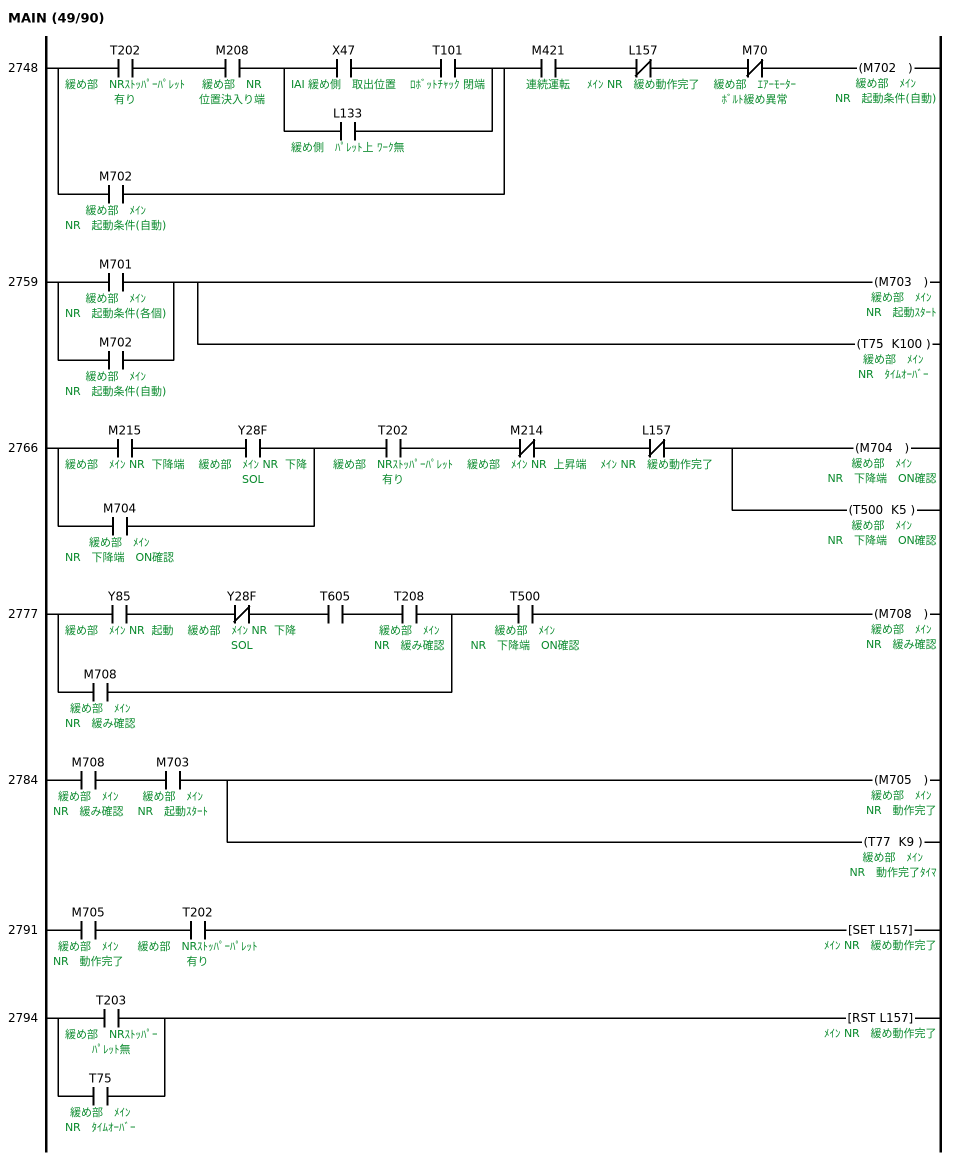
[picture p48: ladder of MAIN, rungs at steps 2748 to 2794]
2748  LD      T202  ; 緩め部　NRｽﾄｯﾊﾟｰﾊﾟﾚｯﾄ有り
      AND     M208  ; 緩め部　NR 位置決入り端
      LD      X47  ; IAI 緩め側　取出位置
      AND     T101  ; ﾛﾎﾞｯﾄﾁｬｯｸ 閉端
      OR      L133  ; 緩め側　ﾊﾟﾚｯﾄ上 ﾜｰｸ無
      ANB
      OR      M702  ; 緩め部　ﾒｲﾝ NR　起動条件(自動)
      AND     M421  ; 連続運転
      ANI     L157  ; ﾒｲﾝ NR　緩め動作完了
      ANI     M70  ; 緩め部　ｴｱｰﾓｰﾀｰ ﾎﾞﾙﾄ緩め異常
      OUT     M702  ; 緩め部　ﾒｲﾝ NR　起動条件(自動)
2759  LD      M701  ; 緩め部　ﾒｲﾝ NR　起動条件(各個)
      OR      M702  ; 緩め部　ﾒｲﾝ NR　起動条件(自動)
      OUT     M703  ; 緩め部　ﾒｲﾝ NR　起動ｽﾀｰﾄ
      OUT     T75 K100  ; 緩め部　ﾒｲﾝ NR　ﾀｲﾑｵｰﾊﾞｰ
2766  LD      M215  ; 緩め部　ﾒｲﾝ NR  下降端
      AND     Y28F  ; 緩め部　ﾒｲﾝ NR  下降 SOL
      OR      M704  ; 緩め部　ﾒｲﾝ NR　下降端　ON確認
      AND     T202  ; 緩め部　NRｽﾄｯﾊﾟｰﾊﾟﾚｯﾄ有り
      ANI     M214  ; 緩め部　ﾒｲﾝ NR  上昇端
      ANI     L157  ; ﾒｲﾝ NR　緩め動作完了
      OUT     M704  ; 緩め部　ﾒｲﾝ NR　下降端　ON確認
      OUT     T500 K5  ; 緩め部　ﾒｲﾝ NR　下降端　ON確認
2777  LD      Y85  ; 緩め部　ﾒｲﾝ NR  起動
      ANI     Y28F  ; 緩め部　ﾒｲﾝ NR  下降 SOL
      AND     T605
      AND     T208  ; 緩め部　ﾒｲﾝ NR　緩み確認
      OR      M708  ; 緩め部　ﾒｲﾝ NR　緩み確認
      AND     T500  ; 緩め部　ﾒｲﾝ NR　下降端　ON確認
      OUT     M708  ; 緩め部　ﾒｲﾝ NR　緩み確認
2784  LD      M708  ; 緩め部　ﾒｲﾝ NR　緩み確認
      AND     M703  ; 緩め部　ﾒｲﾝ NR　起動ｽﾀｰﾄ
      OUT     M705  ; 緩め部　ﾒｲﾝ NR　動作完了
      OUT     T77 K9  ; 緩め部　ﾒｲﾝ NR　動作完了ﾀｲﾏ
2791  LD      M705  ; 緩め部　ﾒｲﾝ NR　動作完了
      AND     T202  ; 緩め部　NRｽﾄｯﾊﾟｰﾊﾟﾚｯﾄ有り
      SET     L157  ; ﾒｲﾝ NR　緩め動作完了
2794  LD      T203  ; 緩め部　NRｽﾄｯﾊﾟｰ ﾊﾟﾚｯﾄ無
      OR      T75  ; 緩め部　ﾒｲﾝ NR　ﾀｲﾑｵｰﾊﾞｰ
      RST     L157  ; ﾒｲﾝ NR　緩め動作完了
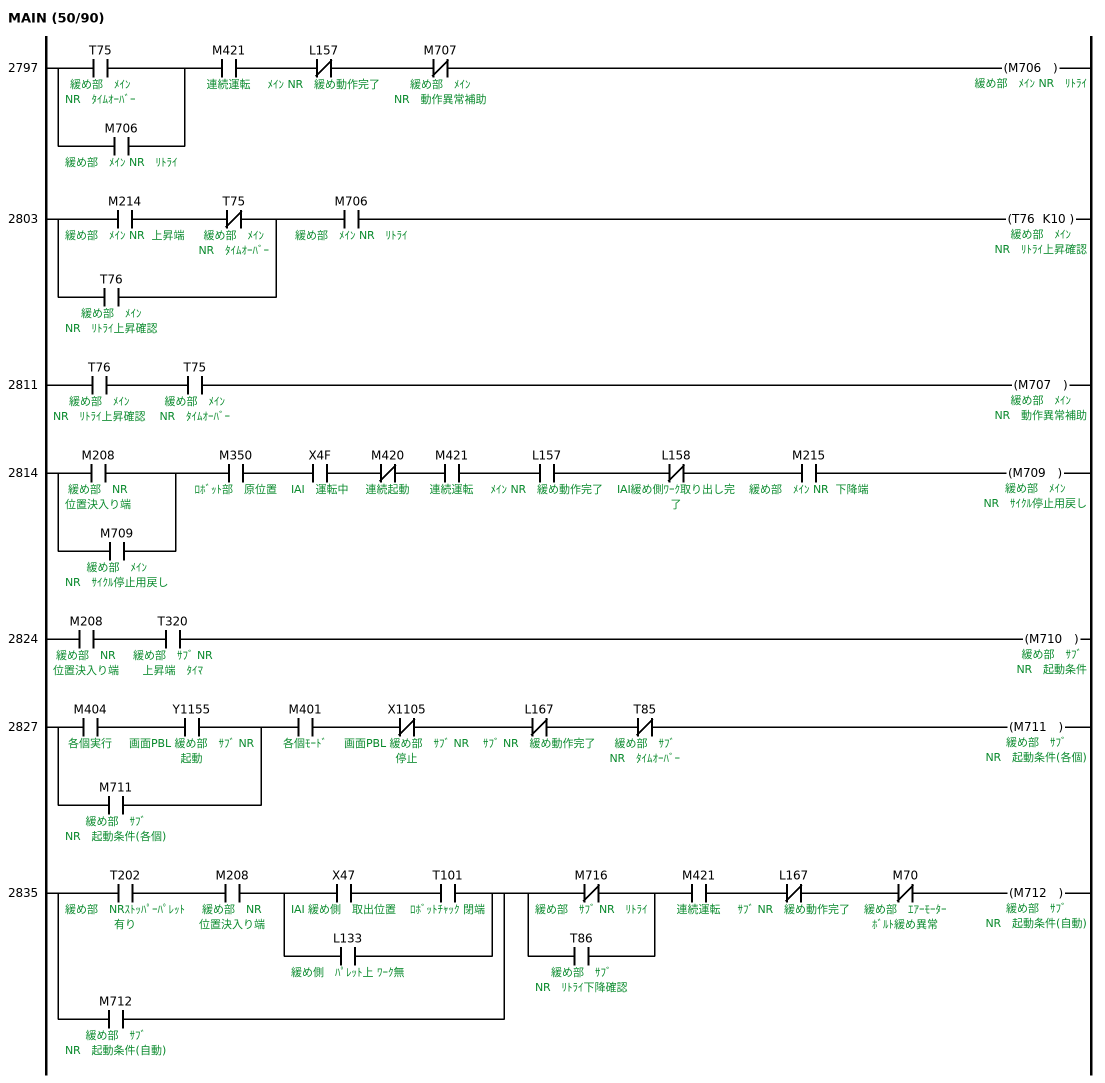
2797  LD      T75  ; 緩め部　ﾒｲﾝ NR　ﾀｲﾑｵｰﾊﾞｰ
      OR      M706  ; 緩め部　ﾒｲﾝ NR　ﾘﾄﾗｲ
      AND     M421  ; 連続運転
      ANI     L157  ; ﾒｲﾝ NR　緩め動作完了
      ANI     M707  ; 緩め部　ﾒｲﾝ NR　動作異常補助
      OUT     M706  ; 緩め部　ﾒｲﾝ NR　ﾘﾄﾗｲ
2803  LD      M214  ; 緩め部　ﾒｲﾝ NR  上昇端
      ANI     T75  ; 緩め部　ﾒｲﾝ NR　ﾀｲﾑｵｰﾊﾞｰ
      OR      T76  ; 緩め部　ﾒｲﾝ NR　ﾘﾄﾗｲ上昇確認
      AND     M706  ; 緩め部　ﾒｲﾝ NR　ﾘﾄﾗｲ
      OUT     T76 K10  ; 緩め部　ﾒｲﾝ NR　ﾘﾄﾗｲ上昇確認
2811  LD      T76  ; 緩め部　ﾒｲﾝ NR　ﾘﾄﾗｲ上昇確認
      AND     T75  ; 緩め部　ﾒｲﾝ NR　ﾀｲﾑｵｰﾊﾞｰ
      OUT     M707  ; 緩め部　ﾒｲﾝ NR　動作異常補助
2814  LD      M208  ; 緩め部　NR 位置決入り端
      OR      M709  ; 緩め部　ﾒｲﾝ NR　ｻｲｸﾙ停止用戻し
      AND     M350  ; ﾛﾎﾞｯﾄ部　原位置
      AND     X4F  ; IAI　運転中
      ANI     M420  ; 連続起動
      AND     M421  ; 連続運転
      AND     L157  ; ﾒｲﾝ NR　緩め動作完了
      ANI     L158  ; IAI緩め側ﾜｰｸ取り出し完了
      AND     M215  ; 緩め部　ﾒｲﾝ NR  下降端
      OUT     M709  ; 緩め部　ﾒｲﾝ NR　ｻｲｸﾙ停止用戻し
2824  LD      M208  ; 緩め部　NR 位置決入り端
      AND     T320  ; 緩め部　ｻﾌﾞ NR  上昇端　ﾀｲﾏ
      OUT     M710  ; 緩め部　ｻﾌﾞ NR　起動条件
2827  LD      M404  ; 各個実行
      AND     Y1155  ; 画面PBL 緩め部　ｻﾌﾞ NR  起動
      OR      M711  ; 緩め部　ｻﾌﾞ NR　起動条件(各個)
      AND     M401  ; 各個ﾓｰﾄﾞ
      ANI     X1105  ; 画面PBL 緩め部　ｻﾌﾞ NR  停止
      ANI     L167  ; ｻﾌﾞ NR　緩め動作完了
      ANI     T85  ; 緩め部　ｻﾌﾞ NR　ﾀｲﾑｵｰﾊﾞｰ
      OUT     M711  ; 緩め部　ｻﾌﾞ NR　起動条件(各個)
2835  LD      T202  ; 緩め部　NRｽﾄｯﾊﾟｰﾊﾟﾚｯﾄ有り
      AND     M208  ; 緩め部　NR 位置決入り端
      LD      X47  ; IAI 緩め側　取出位置
      AND     T101  ; ﾛﾎﾞｯﾄﾁｬｯｸ 閉端
      OR      L133  ; 緩め側　ﾊﾟﾚｯﾄ上 ﾜｰｸ無
      ANB
      OR      M712  ; 緩め部　ｻﾌﾞ NR　起動条件(自動)
      LDI     M716  ; 緩め部　ｻﾌﾞ NR　ﾘﾄﾗｲ
      OR      T86  ; 緩め部　ｻﾌﾞ NR　ﾘﾄﾗｲ下降確認
      ANB
      AND     M421  ; 連続運転
      ANI     L167  ; ｻﾌﾞ NR　緩め動作完了
      ANI     M70  ; 緩め部　ｴｱｰﾓｰﾀｰ ﾎﾞﾙﾄ緩め異常
      OUT     M712  ; 緩め部　ｻﾌﾞ NR　起動条件(自動)
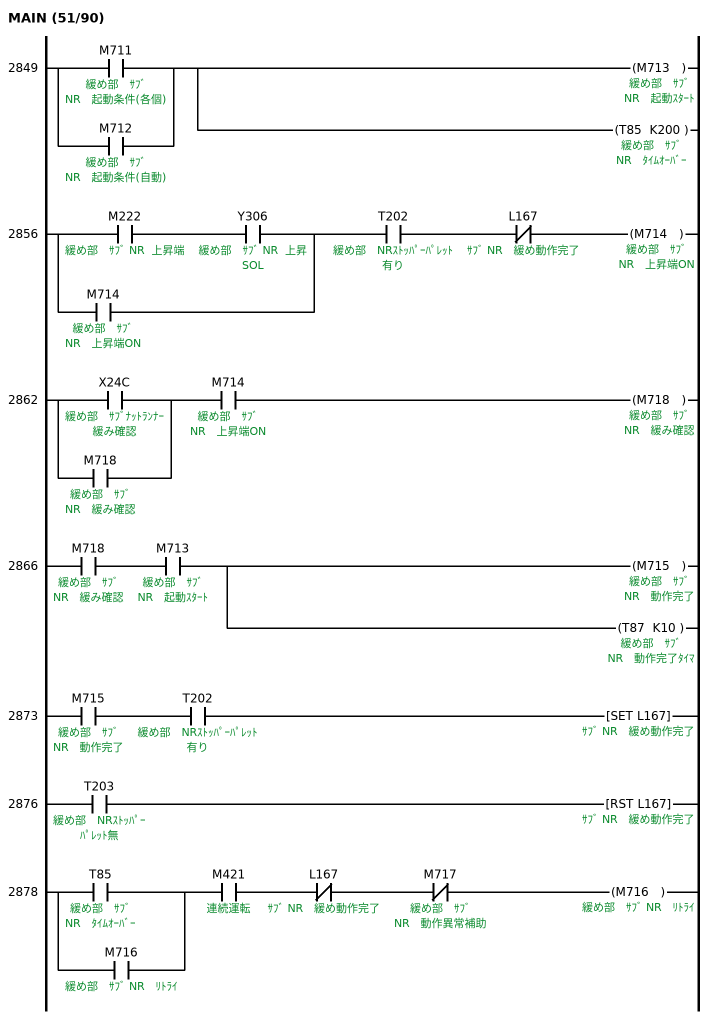
2849  LD      M711  ; 緩め部　ｻﾌﾞ NR　起動条件(各個)
      OR      M712  ; 緩め部　ｻﾌﾞ NR　起動条件(自動)
      OUT     M713  ; 緩め部　ｻﾌﾞ NR　起動ｽﾀｰﾄ
      OUT     T85 K200  ; 緩め部　ｻﾌﾞ NR　ﾀｲﾑｵｰﾊﾞｰ
2856  LD      M222  ; 緩め部　ｻﾌﾞ NR  上昇端
      AND     Y306  ; 緩め部　ｻﾌﾞ NR  上昇 SOL
      OR      M714  ; 緩め部　ｻﾌﾞ NR　上昇端ON
      AND     T202  ; 緩め部　NRｽﾄｯﾊﾟｰﾊﾟﾚｯﾄ有り
      ANI     L167  ; ｻﾌﾞ NR　緩め動作完了
      OUT     M714  ; 緩め部　ｻﾌﾞ NR　上昇端ON
2862  LD      X24C  ; 緩め部　ｻﾌﾞﾅｯﾄﾗﾝﾅｰ 緩み確認
      OR      M718  ; 緩め部　ｻﾌﾞ NR　緩み確認
      AND     M714  ; 緩め部　ｻﾌﾞ NR　上昇端ON
      OUT     M718  ; 緩め部　ｻﾌﾞ NR　緩み確認
2866  LD      M718  ; 緩め部　ｻﾌﾞ NR　緩み確認
      AND     M713  ; 緩め部　ｻﾌﾞ NR　起動ｽﾀｰﾄ
      OUT     M715  ; 緩め部　ｻﾌﾞ NR　動作完了
      OUT     T87 K10  ; 緩め部　ｻﾌﾞ NR　動作完了ﾀｲﾏ
2873  LD      M715  ; 緩め部　ｻﾌﾞ NR　動作完了
      AND     T202  ; 緩め部　NRｽﾄｯﾊﾟｰﾊﾟﾚｯﾄ有り
      SET     L167  ; ｻﾌﾞ NR　緩め動作完了
2876  LD      T203  ; 緩め部　NRｽﾄｯﾊﾟｰ ﾊﾟﾚｯﾄ無
      RST     L167  ; ｻﾌﾞ NR　緩め動作完了
2878  LD      T85  ; 緩め部　ｻﾌﾞ NR　ﾀｲﾑｵｰﾊﾞｰ
      OR      M716  ; 緩め部　ｻﾌﾞ NR　ﾘﾄﾗｲ
      AND     M421  ; 連続運転
      ANI     L167  ; ｻﾌﾞ NR　緩め動作完了
      ANI     M717  ; 緩め部　ｻﾌﾞ NR　動作異常補助
      OUT     M716  ; 緩め部　ｻﾌﾞ NR　ﾘﾄﾗｲ
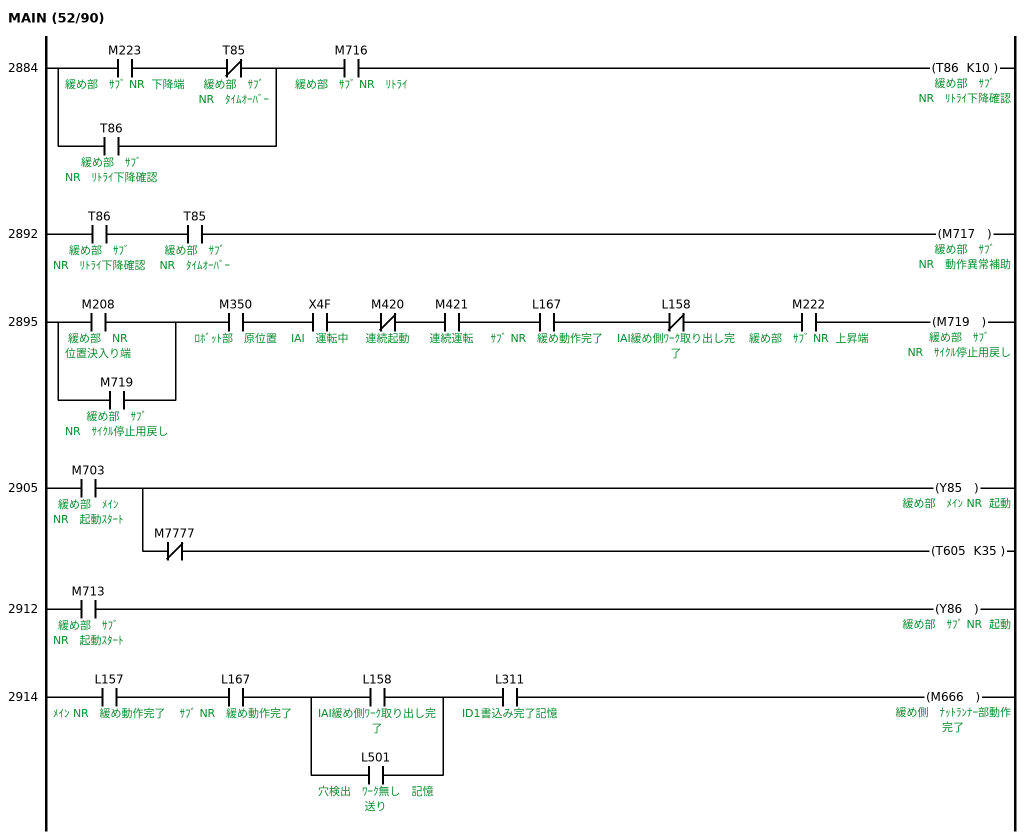
2884  LD      M223  ; 緩め部　ｻﾌﾞ NR  下降端
      ANI     T85  ; 緩め部　ｻﾌﾞ NR　ﾀｲﾑｵｰﾊﾞｰ
      OR      T86  ; 緩め部　ｻﾌﾞ NR　ﾘﾄﾗｲ下降確認
      AND     M716  ; 緩め部　ｻﾌﾞ NR　ﾘﾄﾗｲ
      OUT     T86 K10  ; 緩め部　ｻﾌﾞ NR　ﾘﾄﾗｲ下降確認
2892  LD      T86  ; 緩め部　ｻﾌﾞ NR　ﾘﾄﾗｲ下降確認
      AND     T85  ; 緩め部　ｻﾌﾞ NR　ﾀｲﾑｵｰﾊﾞｰ
      OUT     M717  ; 緩め部　ｻﾌﾞ NR　動作異常補助
2895  LD      M208  ; 緩め部　NR 位置決入り端
      OR      M719  ; 緩め部　ｻﾌﾞ NR　ｻｲｸﾙ停止用戻し
      AND     M350  ; ﾛﾎﾞｯﾄ部　原位置
      AND     X4F  ; IAI　運転中
      ANI     M420  ; 連続起動
      AND     M421  ; 連続運転
      AND     L167  ; ｻﾌﾞ NR　緩め動作完了
      ANI     L158  ; IAI緩め側ﾜｰｸ取り出し完了
      AND     M222  ; 緩め部　ｻﾌﾞ NR  上昇端
      OUT     M719  ; 緩め部　ｻﾌﾞ NR　ｻｲｸﾙ停止用戻し
2905  LD      M703  ; 緩め部　ﾒｲﾝ NR　起動ｽﾀｰﾄ
      OUT     Y85  ; 緩め部　ﾒｲﾝ NR  起動
      ANI     M7777
      OUT     T605 K35
2912  LD      M713  ; 緩め部　ｻﾌﾞ NR　起動ｽﾀｰﾄ
      OUT     Y86  ; 緩め部　ｻﾌﾞ NR  起動
2914  LD      L157  ; ﾒｲﾝ NR　緩め動作完了
      AND     L167  ; ｻﾌﾞ NR　緩め動作完了
      LD      L158  ; IAI緩め側ﾜｰｸ取り出し完了
      OR      L501  ; 穴検出　ﾜｰｸ無し　記憶送り
      ANB
      AND     L311  ; ID1書込み完了記憶
      OUT     M666  ; 緩め側　ﾅｯﾄﾗﾝﾅｰ部動作完了
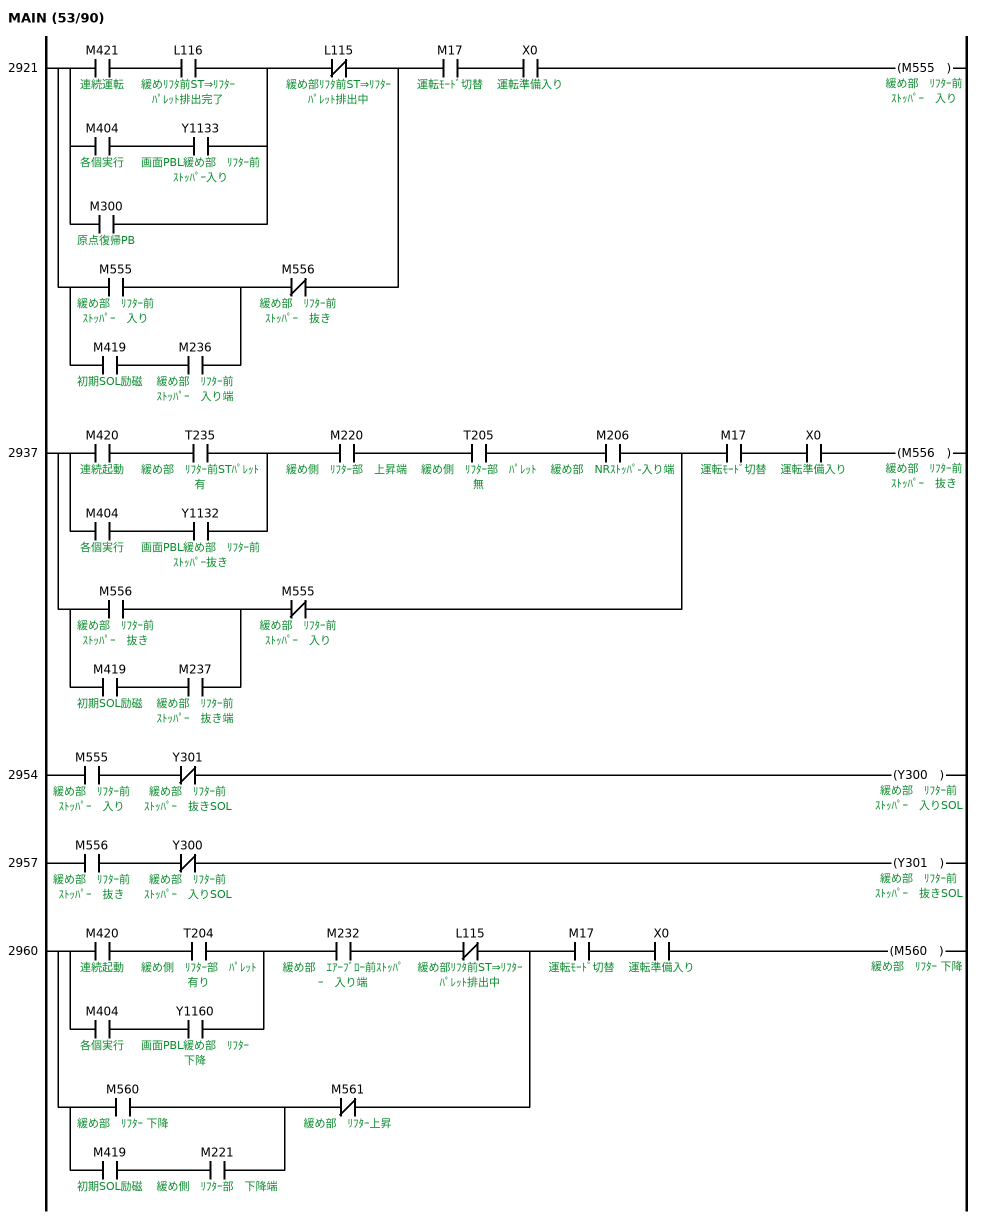
2921  LD      M421  ; 連続運転
      AND     L116  ; 緩めﾘﾌﾀ前ST⇒ﾘﾌﾀｰ ﾊﾟﾚｯﾄ排出完了
      LD      M404  ; 各個実行
      AND     Y1133  ; 画面PBL緩め部　ﾘﾌﾀｰ前 ｽﾄｯﾊﾟｰ入り
      ORB
      OR      M300  ; 原点復帰PB
      ANI     L115  ; 緩め部ﾘﾌﾀ前ST⇒ﾘﾌﾀｰ ﾊﾟﾚｯﾄ排出中
      LD      M555  ; 緩め部　ﾘﾌﾀｰ前  ｽﾄｯﾊﾟｰ　入り
      LD      M419  ; 初期SOL励磁
      AND     M236  ; 緩め部　ﾘﾌﾀｰ前  ｽﾄｯﾊﾟｰ　入り端
      ORB
      ANI     M556  ; 緩め部　ﾘﾌﾀｰ前  ｽﾄｯﾊﾟｰ　抜き
      ORB
      AND     M17  ; 運転ﾓｰﾄﾞ切替
      AND     X0  ; 運転準備入り
      OUT     M555  ; 緩め部　ﾘﾌﾀｰ前  ｽﾄｯﾊﾟｰ　入り
2937  LD      M420  ; 連続起動
      AND     T235  ; 緩め部　ﾘﾌﾀｰ前STﾊﾟﾚｯﾄ有
      LD      M404  ; 各個実行
      AND     Y1132  ; 画面PBL緩め部　ﾘﾌﾀｰ前 ｽﾄｯﾊﾟｰ抜き
      ORB
      AND     M220  ; 緩め側　ﾘﾌﾀｰ部　上昇端
      AND     T205  ; 緩め側　ﾘﾌﾀｰ部　ﾊﾟﾚｯﾄ無
      AND     M206  ; 緩め部　NRｽﾄｯﾊﾟ-入り端
      LD      M556  ; 緩め部　ﾘﾌﾀｰ前  ｽﾄｯﾊﾟｰ　抜き
      LD      M419  ; 初期SOL励磁
      AND     M237  ; 緩め部　ﾘﾌﾀｰ前  ｽﾄｯﾊﾟｰ　抜き端
      ORB
      ANI     M555  ; 緩め部　ﾘﾌﾀｰ前  ｽﾄｯﾊﾟｰ　入り
      ORB
      AND     M17  ; 運転ﾓｰﾄﾞ切替
      AND     X0  ; 運転準備入り
      OUT     M556  ; 緩め部　ﾘﾌﾀｰ前  ｽﾄｯﾊﾟｰ　抜き
2954  LD      M555  ; 緩め部　ﾘﾌﾀｰ前  ｽﾄｯﾊﾟｰ　入り
      ANI     Y301  ; 緩め部　ﾘﾌﾀｰ前  ｽﾄｯﾊﾟｰ　抜きSOL
      OUT     Y300  ; 緩め部　ﾘﾌﾀｰ前  ｽﾄｯﾊﾟｰ　入りSOL
2957  LD      M556  ; 緩め部　ﾘﾌﾀｰ前  ｽﾄｯﾊﾟｰ　抜き
      ANI     Y300  ; 緩め部　ﾘﾌﾀｰ前  ｽﾄｯﾊﾟｰ　入りSOL
      OUT     Y301  ; 緩め部　ﾘﾌﾀｰ前  ｽﾄｯﾊﾟｰ　抜きSOL
2960  LD      M420  ; 連続起動
      AND     T204  ; 緩め側　ﾘﾌﾀｰ部　ﾊﾟﾚｯﾄ有り
      LD      M404  ; 各個実行
      AND     Y1160  ; 画面PBL緩め部　ﾘﾌﾀｰ 下降
      ORB
      AND     M232  ; 緩め部　ｴｱｰﾌﾞﾛｰ前ｽﾄｯﾊﾟｰ　入り端
      ANI     L115  ; 緩め部ﾘﾌﾀ前ST⇒ﾘﾌﾀｰ ﾊﾟﾚｯﾄ排出中
      LD      M560  ; 緩め部　ﾘﾌﾀｰ 下降
      LD      M419  ; 初期SOL励磁
      AND     M221  ; 緩め側　ﾘﾌﾀｰ部　下降端
      ORB
      ANI     M561  ; 緩め部　ﾘﾌﾀｰ上昇
      ORB
      AND     M17  ; 運転ﾓｰﾄﾞ切替
      AND     X0  ; 運転準備入り
      OUT     M560  ; 緩め部　ﾘﾌﾀｰ 下降
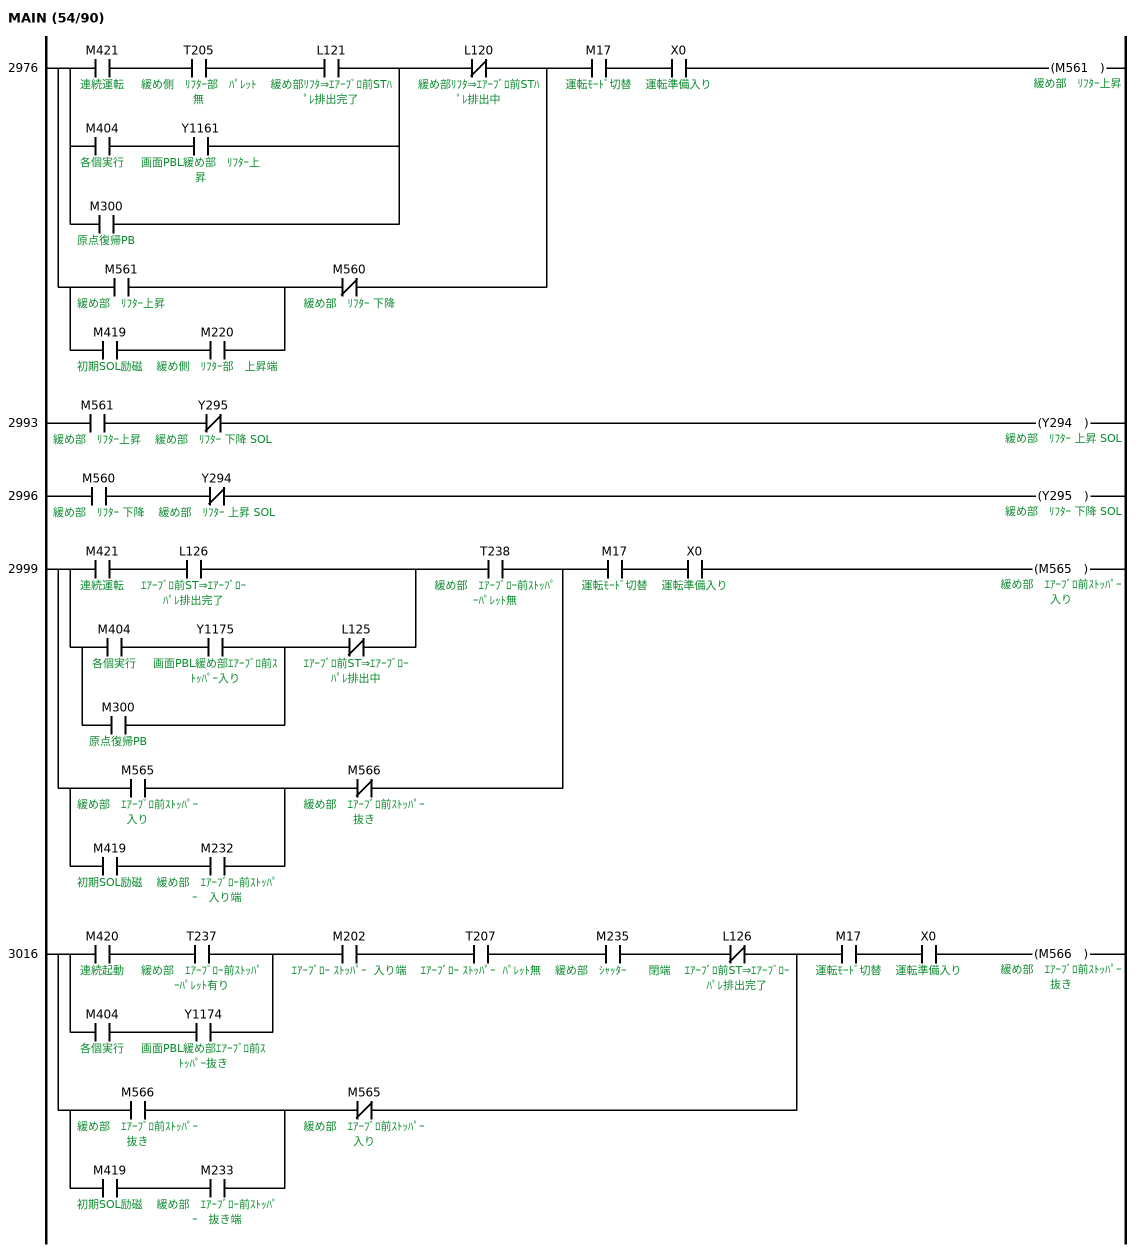
2976  LD      M421  ; 連続運転
      AND     T205  ; 緩め側　ﾘﾌﾀｰ部　ﾊﾟﾚｯﾄ無
      AND     L121  ; 緩め部ﾘﾌﾀ⇒ｴｱｰﾌﾞﾛ前STﾊﾟﾚ排出完了
      LD      M404  ; 各個実行
      AND     Y1161  ; 画面PBL緩め部　ﾘﾌﾀｰ上昇
      ORB
      OR      M300  ; 原点復帰PB
      ANI     L120  ; 緩め部ﾘﾌﾀ⇒ｴｱｰﾌﾞﾛ前STﾊﾟﾚ排出中
      LD      M561  ; 緩め部　ﾘﾌﾀｰ上昇
      LD      M419  ; 初期SOL励磁
      AND     M220  ; 緩め側　ﾘﾌﾀｰ部　上昇端
      ORB
      ANI     M560  ; 緩め部　ﾘﾌﾀｰ 下降
      ORB
      AND     M17  ; 運転ﾓｰﾄﾞ切替
      AND     X0  ; 運転準備入り
      OUT     M561  ; 緩め部　ﾘﾌﾀｰ上昇
2993  LD      M561  ; 緩め部　ﾘﾌﾀｰ上昇
      ANI     Y295  ; 緩め部　ﾘﾌﾀｰ 下降 SOL
      OUT     Y294  ; 緩め部　ﾘﾌﾀｰ 上昇 SOL
2996  LD      M560  ; 緩め部　ﾘﾌﾀｰ 下降
      ANI     Y294  ; 緩め部　ﾘﾌﾀｰ 上昇 SOL
      OUT     Y295  ; 緩め部　ﾘﾌﾀｰ 下降 SOL
2999  LD      M421  ; 連続運転
      AND     L126  ; ｴｱｰﾌﾞﾛ前ST⇒ｴｱｰﾌﾞﾛｰ ﾊﾟﾚ排出完了
      LD      M404  ; 各個実行
      AND     Y1175  ; 画面PBL緩め部ｴｱｰﾌﾞﾛ前ｽﾄｯﾊﾟｰ入り
      OR      M300  ; 原点復帰PB
      ANI     L125  ; ｴｱｰﾌﾞﾛ前ST⇒ｴｱｰﾌﾞﾛｰ ﾊﾟﾚ排出中
      ORB
      AND     T238  ; 緩め部　ｴｱｰﾌﾞﾛｰ前ｽﾄｯﾊﾟｰﾊﾟﾚｯﾄ無
      LD      M565  ; 緩め部　ｴｱｰﾌﾞﾛ前ｽﾄｯﾊﾟｰ　入り
      LD      M419  ; 初期SOL励磁
      AND     M232  ; 緩め部　ｴｱｰﾌﾞﾛｰ前ｽﾄｯﾊﾟｰ　入り端
      ORB
      ANI     M566  ; 緩め部　ｴｱｰﾌﾞﾛ前ｽﾄｯﾊﾟｰ　抜き
      ORB
      AND     M17  ; 運転ﾓｰﾄﾞ切替
      AND     X0  ; 運転準備入り
      OUT     M565  ; 緩め部　ｴｱｰﾌﾞﾛ前ｽﾄｯﾊﾟｰ　入り
3016  LD      M420  ; 連続起動
      AND     T237  ; 緩め部　ｴｱｰﾌﾞﾛｰ前ｽﾄｯﾊﾟｰﾊﾟﾚｯﾄ有り
      LD      M404  ; 各個実行
      AND     Y1174  ; 画面PBL緩め部ｴｱｰﾌﾞﾛ前ｽﾄｯﾊﾟｰ抜き
      ORB
      AND     M202  ; ｴｱｰﾌﾞﾛｰ ｽﾄｯﾊﾟｰ  入り端
      AND     T207  ; ｴｱｰﾌﾞﾛｰ ｽﾄｯﾊﾟｰ  ﾊﾟﾚｯﾄ無
      AND     M235  ; 緩め部　ｼｬｯﾀｰ　　閉端
      ANI     L126  ; ｴｱｰﾌﾞﾛ前ST⇒ｴｱｰﾌﾞﾛｰ ﾊﾟﾚ排出完了
      LD      M566  ; 緩め部　ｴｱｰﾌﾞﾛ前ｽﾄｯﾊﾟｰ　抜き
      LD      M419  ; 初期SOL励磁
      AND     M233  ; 緩め部　ｴｱｰﾌﾞﾛｰ前ｽﾄｯﾊﾟｰ　抜き端
      ORB
      ANI     M565  ; 緩め部　ｴｱｰﾌﾞﾛ前ｽﾄｯﾊﾟｰ　入り
      ORB
      AND     M17  ; 運転ﾓｰﾄﾞ切替
      AND     X0  ; 運転準備入り
      OUT     M566  ; 緩め部　ｴｱｰﾌﾞﾛ前ｽﾄｯﾊﾟｰ　抜き
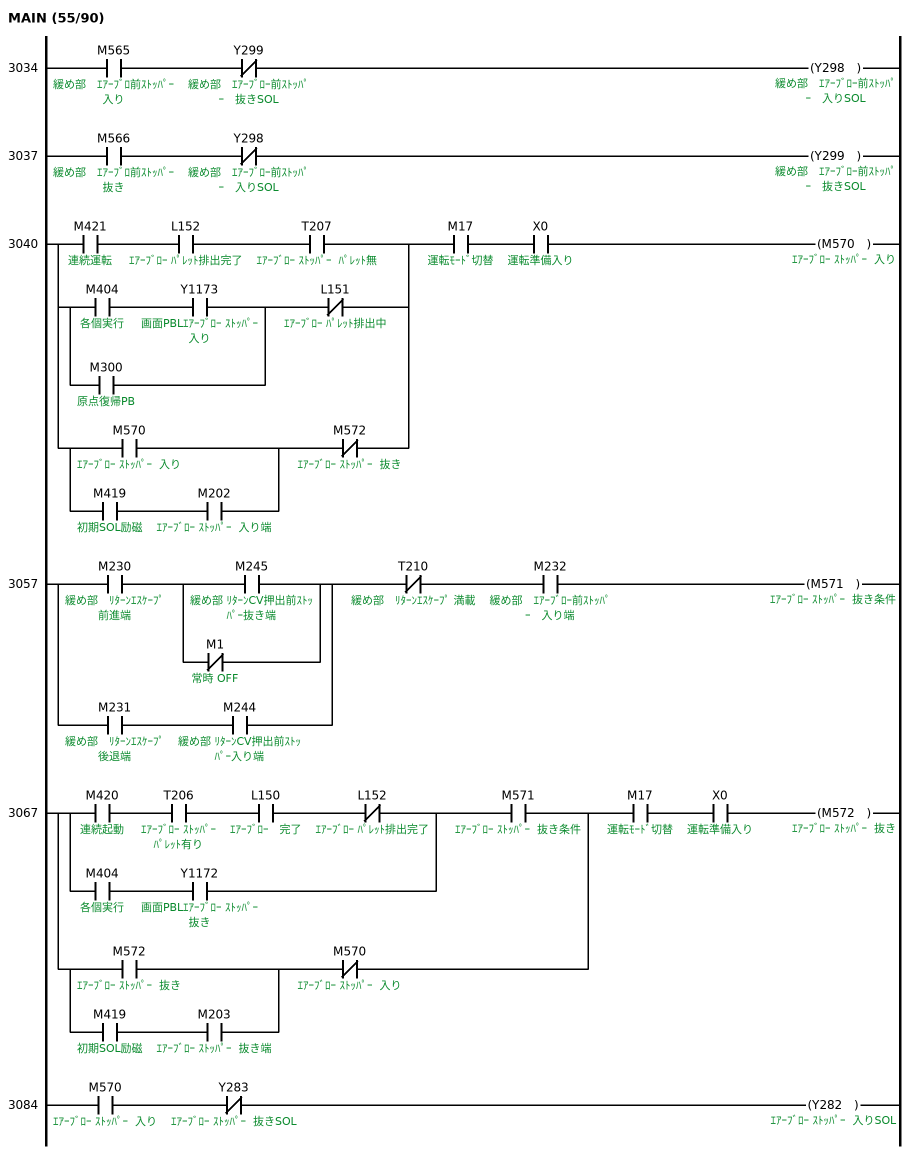
3034  LD      M565  ; 緩め部　ｴｱｰﾌﾞﾛ前ｽﾄｯﾊﾟｰ　入り
      ANI     Y299  ; 緩め部　ｴｱｰﾌﾞﾛｰ前ｽﾄｯﾊﾟｰ　抜きSOL
      OUT     Y298  ; 緩め部　ｴｱｰﾌﾞﾛｰ前ｽﾄｯﾊﾟｰ　入りSOL
3037  LD      M566  ; 緩め部　ｴｱｰﾌﾞﾛ前ｽﾄｯﾊﾟｰ　抜き
      ANI     Y298  ; 緩め部　ｴｱｰﾌﾞﾛｰ前ｽﾄｯﾊﾟｰ　入りSOL
      OUT     Y299  ; 緩め部　ｴｱｰﾌﾞﾛｰ前ｽﾄｯﾊﾟｰ　抜きSOL
3040  LD      M421  ; 連続運転
      AND     L152  ; ｴｱｰﾌﾞﾛｰ ﾊﾟﾚｯﾄ排出完了
      AND     T207  ; ｴｱｰﾌﾞﾛｰ ｽﾄｯﾊﾟｰ  ﾊﾟﾚｯﾄ無
      LD      M404  ; 各個実行
      AND     Y1173  ; 画面PBLｴｱｰﾌﾞﾛｰ ｽﾄｯﾊﾟｰ  入り
      OR      M300  ; 原点復帰PB
      ANI     L151  ; ｴｱｰﾌﾞﾛｰ ﾊﾟﾚｯﾄ排出中
      ORB
      LD      M570  ; ｴｱｰﾌﾞﾛｰ ｽﾄｯﾊﾟｰ  入り
      LD      M419  ; 初期SOL励磁
      AND     M202  ; ｴｱｰﾌﾞﾛｰ ｽﾄｯﾊﾟｰ  入り端
      ORB
      ANI     M572  ; ｴｱｰﾌﾞﾛｰ ｽﾄｯﾊﾟｰ  抜き
      ORB
      AND     M17  ; 運転ﾓｰﾄﾞ切替
      AND     X0  ; 運転準備入り
      OUT     M570  ; ｴｱｰﾌﾞﾛｰ ｽﾄｯﾊﾟｰ  入り
3057  LD      M230  ; 緩め部　ﾘﾀｰﾝｴｽｹｰﾌﾟ 前進端
      LD      M245  ; 緩め部 ﾘﾀｰﾝCV押出前ｽﾄｯﾊﾟｰ抜き端
      ORI     M1  ; 常時 OFF
      ANB
      LD      M231  ; 緩め部　ﾘﾀｰﾝｴｽｹｰﾌﾟ 後退端
      AND     M244  ; 緩め部 ﾘﾀｰﾝCV押出前ｽﾄｯﾊﾟｰ入り端
      ORB
      ANI     T210  ; 緩め部　ﾘﾀｰﾝｴｽｹｰﾌﾟ 満載
      AND     M232  ; 緩め部　ｴｱｰﾌﾞﾛｰ前ｽﾄｯﾊﾟｰ　入り端
      OUT     M571  ; ｴｱｰﾌﾞﾛｰ ｽﾄｯﾊﾟｰ  抜き条件
3067  LD      M420  ; 連続起動
      AND     T206  ; ｴｱｰﾌﾞﾛｰ ｽﾄｯﾊﾟｰ  ﾊﾟﾚｯﾄ有り
      AND     L150  ; ｴｱｰﾌﾞﾛｰ　完了
      ANI     L152  ; ｴｱｰﾌﾞﾛｰ ﾊﾟﾚｯﾄ排出完了
      LD      M404  ; 各個実行
      AND     Y1172  ; 画面PBLｴｱｰﾌﾞﾛｰ ｽﾄｯﾊﾟｰ  抜き
      ORB
      AND     M571  ; ｴｱｰﾌﾞﾛｰ ｽﾄｯﾊﾟｰ  抜き条件
      LD      M572  ; ｴｱｰﾌﾞﾛｰ ｽﾄｯﾊﾟｰ  抜き
      LD      M419  ; 初期SOL励磁
      AND     M203  ; ｴｱｰﾌﾞﾛｰ ｽﾄｯﾊﾟｰ  抜き端
      ORB
      ANI     M570  ; ｴｱｰﾌﾞﾛｰ ｽﾄｯﾊﾟｰ  入り
      ORB
      AND     M17  ; 運転ﾓｰﾄﾞ切替
      AND     X0  ; 運転準備入り
      OUT     M572  ; ｴｱｰﾌﾞﾛｰ ｽﾄｯﾊﾟｰ  抜き
3084  LD      M570  ; ｴｱｰﾌﾞﾛｰ ｽﾄｯﾊﾟｰ  入り
      ANI     Y283  ; ｴｱｰﾌﾞﾛｰ ｽﾄｯﾊﾟｰ  抜きSOL
      OUT     Y282  ; ｴｱｰﾌﾞﾛｰ ｽﾄｯﾊﾟｰ  入りSOL
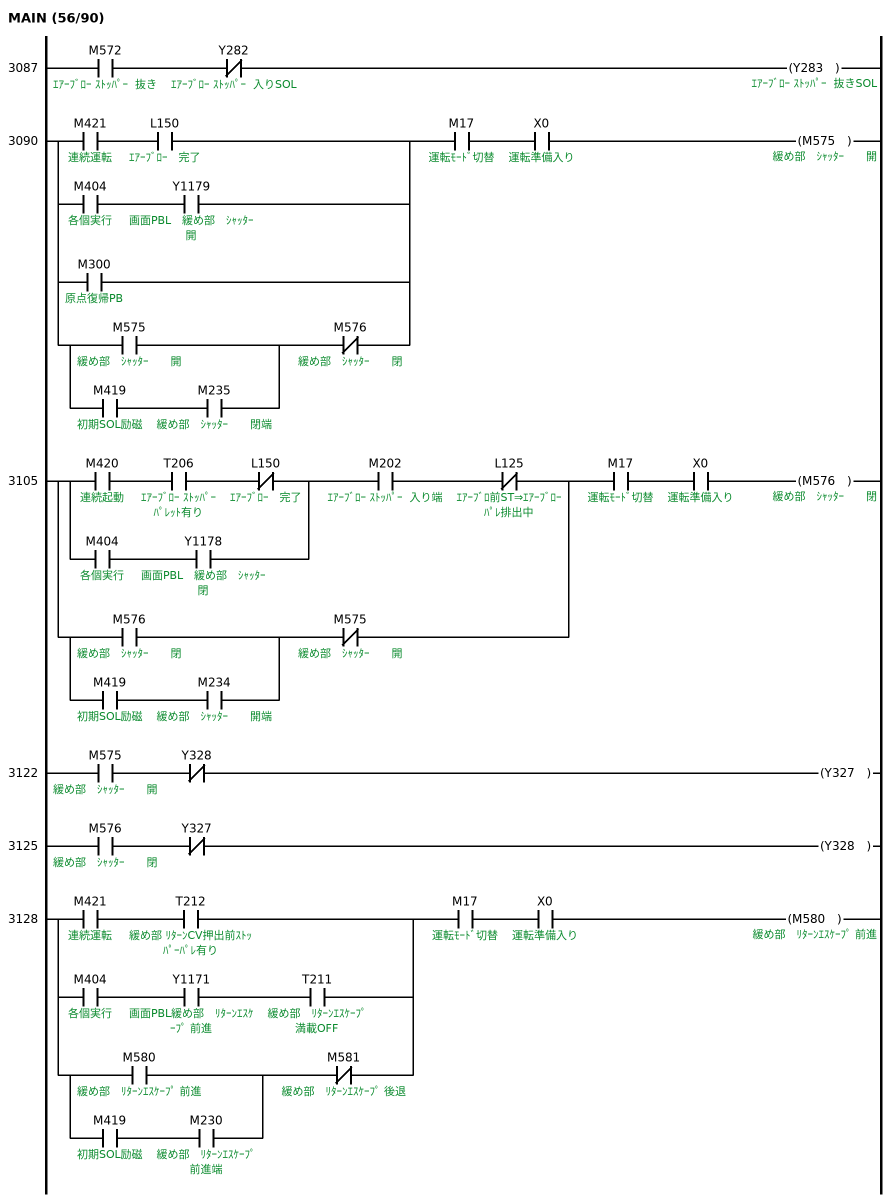
3087  LD      M572  ; ｴｱｰﾌﾞﾛｰ ｽﾄｯﾊﾟｰ  抜き
      ANI     Y282  ; ｴｱｰﾌﾞﾛｰ ｽﾄｯﾊﾟｰ  入りSOL
      OUT     Y283  ; ｴｱｰﾌﾞﾛｰ ｽﾄｯﾊﾟｰ  抜きSOL
3090  LD      M421  ; 連続運転
      AND     L150  ; ｴｱｰﾌﾞﾛｰ　完了
      LD      M404  ; 各個実行
      AND     Y1179  ; 画面PBL　緩め部　ｼｬｯﾀｰ　　開
      ORB
      OR      M300  ; 原点復帰PB
      LD      M575  ; 緩め部　ｼｬｯﾀｰ　　開
      LD      M419  ; 初期SOL励磁
      AND     M235  ; 緩め部　ｼｬｯﾀｰ　　閉端
      ORB
      ANI     M576  ; 緩め部　ｼｬｯﾀｰ　　閉
      ORB
      AND     M17  ; 運転ﾓｰﾄﾞ切替
      AND     X0  ; 運転準備入り
      OUT     M575  ; 緩め部　ｼｬｯﾀｰ　　開
3105  LD      M420  ; 連続起動
      AND     T206  ; ｴｱｰﾌﾞﾛｰ ｽﾄｯﾊﾟｰ  ﾊﾟﾚｯﾄ有り
      ANI     L150  ; ｴｱｰﾌﾞﾛｰ　完了
      LD      M404  ; 各個実行
      AND     Y1178  ; 画面PBL　緩め部　ｼｬｯﾀｰ　　閉
      ORB
      AND     M202  ; ｴｱｰﾌﾞﾛｰ ｽﾄｯﾊﾟｰ  入り端
      ANI     L125  ; ｴｱｰﾌﾞﾛ前ST⇒ｴｱｰﾌﾞﾛｰ ﾊﾟﾚ排出中
      LD      M576  ; 緩め部　ｼｬｯﾀｰ　　閉
      LD      M419  ; 初期SOL励磁
      AND     M234  ; 緩め部　ｼｬｯﾀｰ　　開端
      ORB
      ANI     M575  ; 緩め部　ｼｬｯﾀｰ　　開
      ORB
      AND     M17  ; 運転ﾓｰﾄﾞ切替
      AND     X0  ; 運転準備入り
      OUT     M576  ; 緩め部　ｼｬｯﾀｰ　　閉
3122  LD      M575  ; 緩め部　ｼｬｯﾀｰ　　開
      ANI     Y328
      OUT     Y327
3125  LD      M576  ; 緩め部　ｼｬｯﾀｰ　　閉
      ANI     Y327
      OUT     Y328
3128  LD      M421  ; 連続運転
      AND     T212  ; 緩め部 ﾘﾀｰﾝCV押出前ｽﾄｯﾊﾟｰﾊﾟﾚ有り
      LD      M404  ; 各個実行
      AND     Y1171  ; 画面PBL緩め部　ﾘﾀｰﾝｴｽｹｰﾌﾟ 前進
      AND     T211  ; 緩め部　ﾘﾀｰﾝｴｽｹｰﾌﾟ 満載OFF
      ORB
      LD      M580  ; 緩め部　ﾘﾀｰﾝｴｽｹｰﾌﾟ 前進
      LD      M419  ; 初期SOL励磁
      AND     M230  ; 緩め部　ﾘﾀｰﾝｴｽｹｰﾌﾟ 前進端
      ORB
      ANI     M581  ; 緩め部　ﾘﾀｰﾝｴｽｹｰﾌﾟ 後退
      ORB
      AND     M17  ; 運転ﾓｰﾄﾞ切替
      AND     X0  ; 運転準備入り
      OUT     M580  ; 緩め部　ﾘﾀｰﾝｴｽｹｰﾌﾟ 前進
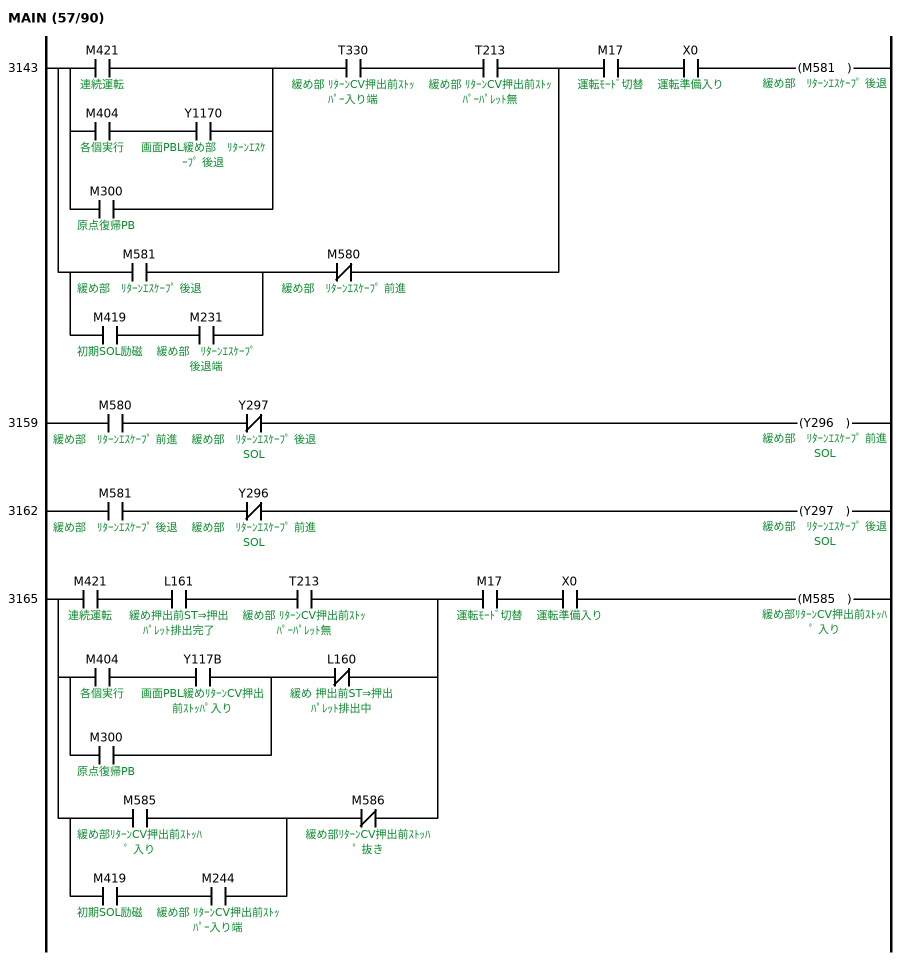
3143  LD      M421  ; 連続運転
      LD      M404  ; 各個実行
      AND     Y1170  ; 画面PBL緩め部　ﾘﾀｰﾝｴｽｹｰﾌﾟ 後退
      ORB
      OR      M300  ; 原点復帰PB
      AND     T330  ; 緩め部 ﾘﾀｰﾝCV押出前ｽﾄｯﾊﾟｰ入り端
      AND     T213  ; 緩め部 ﾘﾀｰﾝCV押出前ｽﾄｯﾊﾟｰﾊﾟﾚｯﾄ無
      LD      M581  ; 緩め部　ﾘﾀｰﾝｴｽｹｰﾌﾟ 後退
      LD      M419  ; 初期SOL励磁
      AND     M231  ; 緩め部　ﾘﾀｰﾝｴｽｹｰﾌﾟ 後退端
      ORB
      ANI     M580  ; 緩め部　ﾘﾀｰﾝｴｽｹｰﾌﾟ 前進
      ORB
      AND     M17  ; 運転ﾓｰﾄﾞ切替
      AND     X0  ; 運転準備入り
      OUT     M581  ; 緩め部　ﾘﾀｰﾝｴｽｹｰﾌﾟ 後退
3159  LD      M580  ; 緩め部　ﾘﾀｰﾝｴｽｹｰﾌﾟ 前進
      ANI     Y297  ; 緩め部　ﾘﾀｰﾝｴｽｹｰﾌﾟ 後退 SOL
      OUT     Y296  ; 緩め部　ﾘﾀｰﾝｴｽｹｰﾌﾟ 前進 SOL
3162  LD      M581  ; 緩め部　ﾘﾀｰﾝｴｽｹｰﾌﾟ 後退
      ANI     Y296  ; 緩め部　ﾘﾀｰﾝｴｽｹｰﾌﾟ 前進 SOL
      OUT     Y297  ; 緩め部　ﾘﾀｰﾝｴｽｹｰﾌﾟ 後退 SOL
3165  LD      M421  ; 連続運転
      AND     L161  ; 緩め押出前ST⇒押出 ﾊﾟﾚｯﾄ排出完了
      AND     T213  ; 緩め部 ﾘﾀｰﾝCV押出前ｽﾄｯﾊﾟｰﾊﾟﾚｯﾄ無
      LD      M404  ; 各個実行
      AND     Y117B  ; 画面PBL緩めﾘﾀｰﾝCV押出前ｽﾄｯﾊﾟ入り
      OR      M300  ; 原点復帰PB
      ANI     L160  ; 緩め 押出前ST⇒押出 ﾊﾟﾚｯﾄ排出中
      ORB
      LD      M585  ; 緩め部ﾘﾀｰﾝCV押出前ｽﾄｯﾊﾟ 入り
      LD      M419  ; 初期SOL励磁
      AND     M244  ; 緩め部 ﾘﾀｰﾝCV押出前ｽﾄｯﾊﾟｰ入り端
      ORB
      ANI     M586  ; 緩め部ﾘﾀｰﾝCV押出前ｽﾄｯﾊﾟ 抜き
      ORB
      AND     M17  ; 運転ﾓｰﾄﾞ切替
      AND     X0  ; 運転準備入り
      OUT     M585  ; 緩め部ﾘﾀｰﾝCV押出前ｽﾄｯﾊﾟ 入り
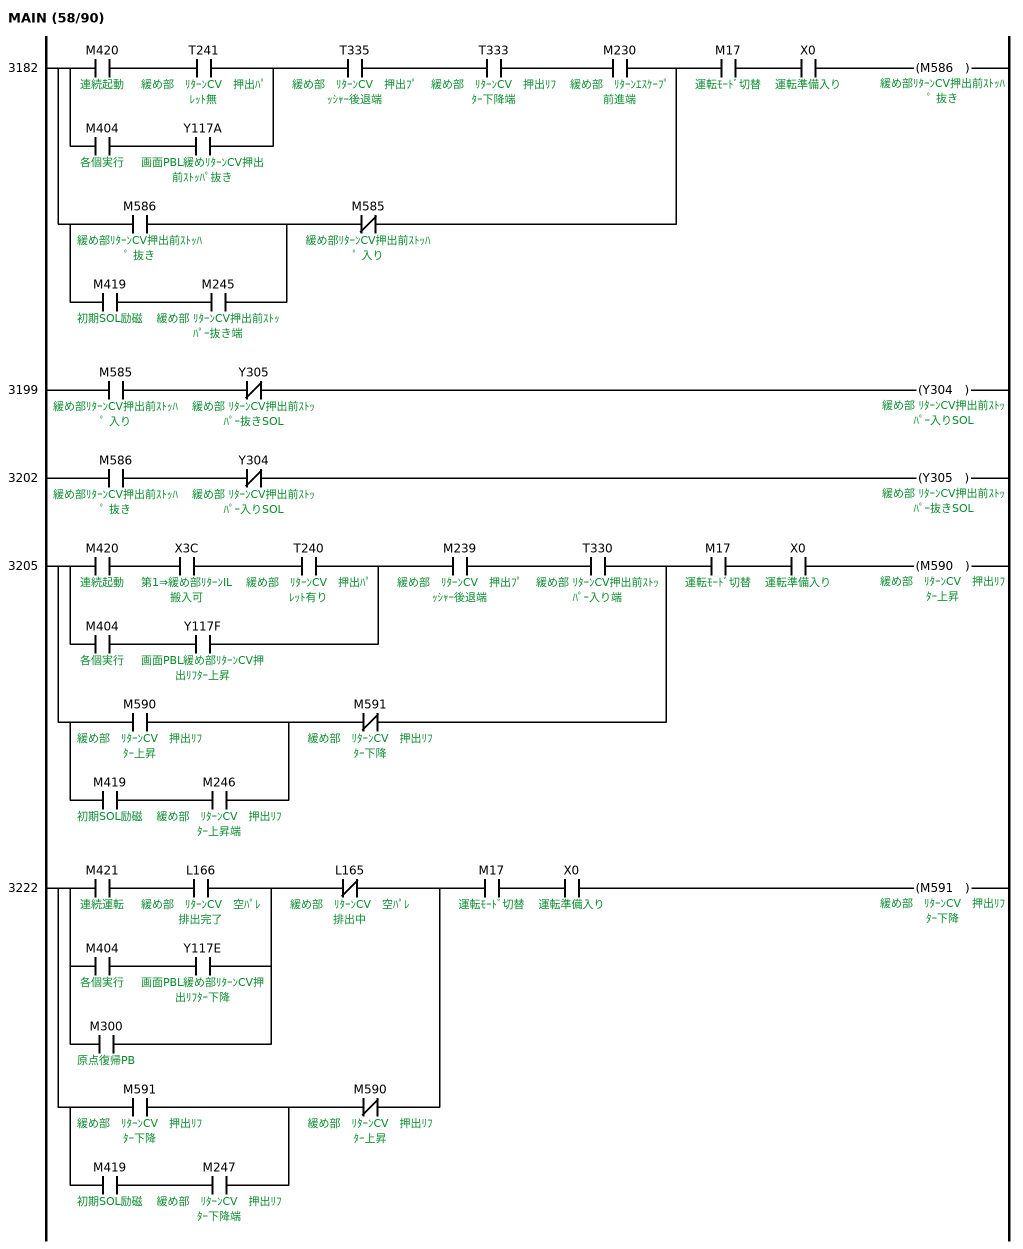
3182  LD      M420  ; 連続起動
      AND     T241  ; 緩め部　ﾘﾀｰﾝCV　押出ﾊﾟﾚｯﾄ無
      LD      M404  ; 各個実行
      AND     Y117A  ; 画面PBL緩めﾘﾀｰﾝCV押出前ｽﾄｯﾊﾟ抜き
      ORB
      AND     T335  ; 緩め部　ﾘﾀｰﾝCV　押出ﾌﾟｯｼｬｰ後退端
      AND     T333  ; 緩め部　ﾘﾀｰﾝCV　押出ﾘﾌﾀｰ下降端
      AND     M230  ; 緩め部　ﾘﾀｰﾝｴｽｹｰﾌﾟ 前進端
      LD      M586  ; 緩め部ﾘﾀｰﾝCV押出前ｽﾄｯﾊﾟ 抜き
      LD      M419  ; 初期SOL励磁
      AND     M245  ; 緩め部 ﾘﾀｰﾝCV押出前ｽﾄｯﾊﾟｰ抜き端
      ORB
      ANI     M585  ; 緩め部ﾘﾀｰﾝCV押出前ｽﾄｯﾊﾟ 入り
      ORB
      AND     M17  ; 運転ﾓｰﾄﾞ切替
      AND     X0  ; 運転準備入り
      OUT     M586  ; 緩め部ﾘﾀｰﾝCV押出前ｽﾄｯﾊﾟ 抜き
3199  LD      M585  ; 緩め部ﾘﾀｰﾝCV押出前ｽﾄｯﾊﾟ 入り
      ANI     Y305  ; 緩め部 ﾘﾀｰﾝCV押出前ｽﾄｯﾊﾟｰ抜きSOL
      OUT     Y304  ; 緩め部 ﾘﾀｰﾝCV押出前ｽﾄｯﾊﾟｰ入りSOL
3202  LD      M586  ; 緩め部ﾘﾀｰﾝCV押出前ｽﾄｯﾊﾟ 抜き
      ANI     Y304  ; 緩め部 ﾘﾀｰﾝCV押出前ｽﾄｯﾊﾟｰ入りSOL
      OUT     Y305  ; 緩め部 ﾘﾀｰﾝCV押出前ｽﾄｯﾊﾟｰ抜きSOL
3205  LD      M420  ; 連続起動
      AND     X3C  ; 第1⇒緩め部ﾘﾀｰﾝIL 搬入可
      AND     T240  ; 緩め部　ﾘﾀｰﾝCV　押出ﾊﾟﾚｯﾄ有り
      LD      M404  ; 各個実行
      AND     Y117F  ; 画面PBL緩め部ﾘﾀｰﾝCV押出ﾘﾌﾀｰ上昇
      ORB
      AND     M239  ; 緩め部　ﾘﾀｰﾝCV　押出ﾌﾟｯｼｬｰ後退端
      AND     T330  ; 緩め部 ﾘﾀｰﾝCV押出前ｽﾄｯﾊﾟｰ入り端
      LD      M590  ; 緩め部　ﾘﾀｰﾝCV　押出ﾘﾌﾀｰ上昇
      LD      M419  ; 初期SOL励磁
      AND     M246  ; 緩め部　ﾘﾀｰﾝCV　押出ﾘﾌﾀｰ上昇端
      ORB
      ANI     M591  ; 緩め部　ﾘﾀｰﾝCV　押出ﾘﾌﾀｰ下降
      ORB
      AND     M17  ; 運転ﾓｰﾄﾞ切替
      AND     X0  ; 運転準備入り
      OUT     M590  ; 緩め部　ﾘﾀｰﾝCV　押出ﾘﾌﾀｰ上昇
3222  LD      M421  ; 連続運転
      AND     L166  ; 緩め部　ﾘﾀｰﾝCV　空ﾊﾟﾚ排出完了
      LD      M404  ; 各個実行
      AND     Y117E  ; 画面PBL緩め部ﾘﾀｰﾝCV押出ﾘﾌﾀｰ下降
      ORB
      OR      M300  ; 原点復帰PB
      ANI     L165  ; 緩め部　ﾘﾀｰﾝCV　空ﾊﾟﾚ排出中
      LD      M591  ; 緩め部　ﾘﾀｰﾝCV　押出ﾘﾌﾀｰ下降
      LD      M419  ; 初期SOL励磁
      AND     M247  ; 緩め部　ﾘﾀｰﾝCV　押出ﾘﾌﾀｰ下降端
      ORB
      ANI     M590  ; 緩め部　ﾘﾀｰﾝCV　押出ﾘﾌﾀｰ上昇
      ORB
      AND     M17  ; 運転ﾓｰﾄﾞ切替
      AND     X0  ; 運転準備入り
      OUT     M591  ; 緩め部　ﾘﾀｰﾝCV　押出ﾘﾌﾀｰ下降
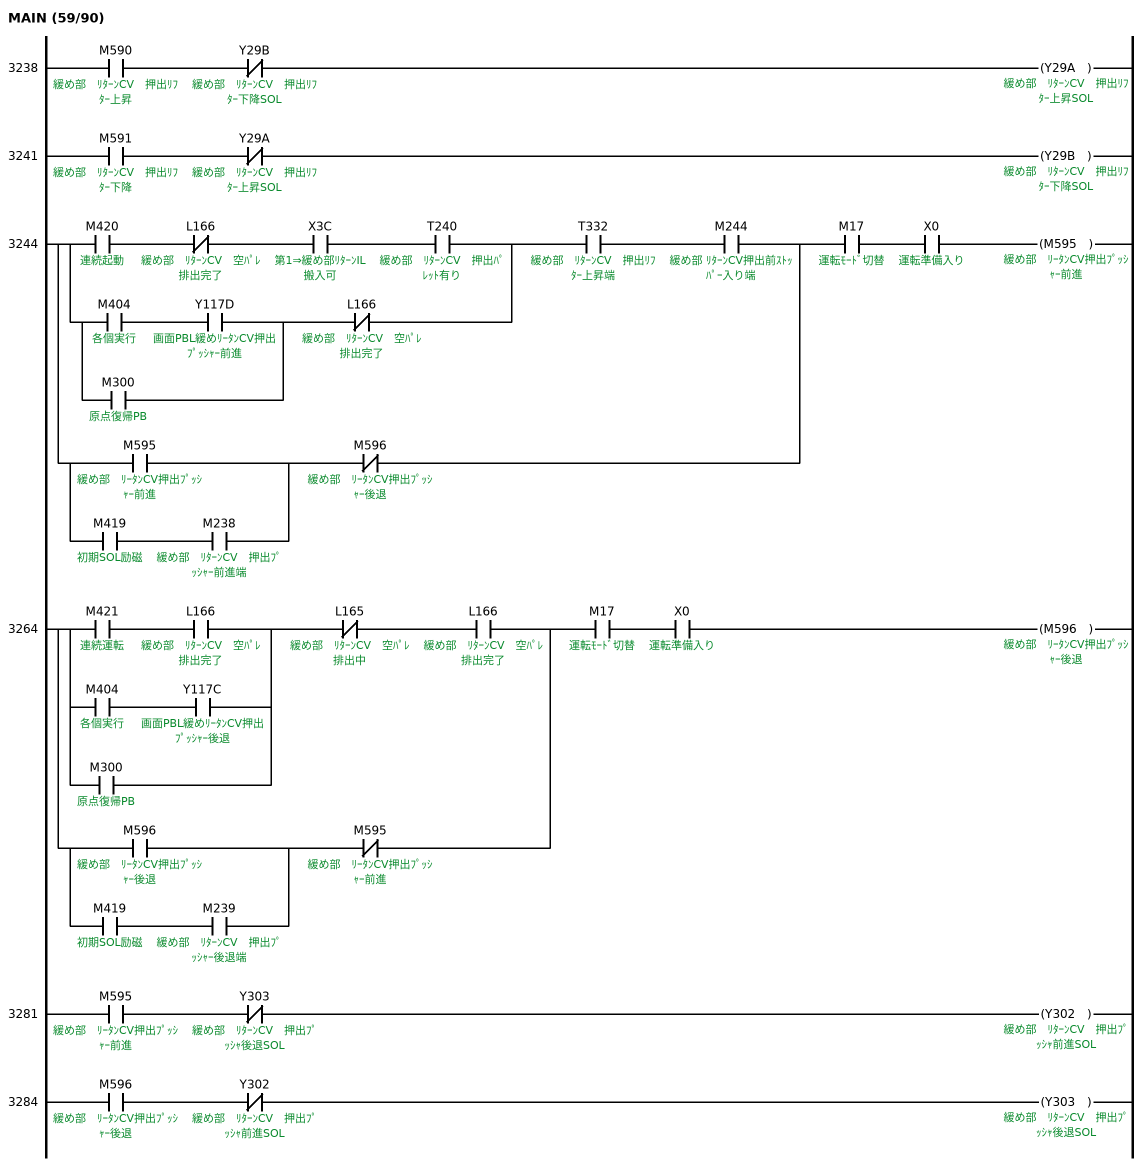
3238  LD      M590  ; 緩め部　ﾘﾀｰﾝCV　押出ﾘﾌﾀｰ上昇
      ANI     Y29B  ; 緩め部　ﾘﾀｰﾝCV　押出ﾘﾌﾀｰ下降SOL
      OUT     Y29A  ; 緩め部　ﾘﾀｰﾝCV　押出ﾘﾌﾀｰ上昇SOL
3241  LD      M591  ; 緩め部　ﾘﾀｰﾝCV　押出ﾘﾌﾀｰ下降
      ANI     Y29A  ; 緩め部　ﾘﾀｰﾝCV　押出ﾘﾌﾀｰ上昇SOL
      OUT     Y29B  ; 緩め部　ﾘﾀｰﾝCV　押出ﾘﾌﾀｰ下降SOL
3244  LD      M420  ; 連続起動
      ANI     L166  ; 緩め部　ﾘﾀｰﾝCV　空ﾊﾟﾚ排出完了
      AND     X3C  ; 第1⇒緩め部ﾘﾀｰﾝIL 搬入可
      AND     T240  ; 緩め部　ﾘﾀｰﾝCV　押出ﾊﾟﾚｯﾄ有り
      LD      M404  ; 各個実行
      AND     Y117D  ; 画面PBL緩めﾘｰﾀﾝCV押出ﾌﾟｯｼｬｰ前進
      OR      M300  ; 原点復帰PB
      ANI     L166  ; 緩め部　ﾘﾀｰﾝCV　空ﾊﾟﾚ排出完了
      ORB
      AND     T332  ; 緩め部　ﾘﾀｰﾝCV　押出ﾘﾌﾀｰ上昇端
      AND     M244  ; 緩め部 ﾘﾀｰﾝCV押出前ｽﾄｯﾊﾟｰ入り端
      LD      M595  ; 緩め部　ﾘｰﾀﾝCV押出ﾌﾟｯｼｬｰ前進
      LD      M419  ; 初期SOL励磁
      AND     M238  ; 緩め部　ﾘﾀｰﾝCV　押出ﾌﾟｯｼｬｰ前進端
      ORB
      ANI     M596  ; 緩め部　ﾘｰﾀﾝCV押出ﾌﾟｯｼｬｰ後退
      ORB
      AND     M17  ; 運転ﾓｰﾄﾞ切替
      AND     X0  ; 運転準備入り
      OUT     M595  ; 緩め部　ﾘｰﾀﾝCV押出ﾌﾟｯｼｬｰ前進
3264  LD      M421  ; 連続運転
      AND     L166  ; 緩め部　ﾘﾀｰﾝCV　空ﾊﾟﾚ排出完了
      LD      M404  ; 各個実行
      AND     Y117C  ; 画面PBL緩めﾘｰﾀﾝCV押出ﾌﾟｯｼｬｰ後退
      ORB
      OR      M300  ; 原点復帰PB
      ANI     L165  ; 緩め部　ﾘﾀｰﾝCV　空ﾊﾟﾚ排出中
      AND     L166  ; 緩め部　ﾘﾀｰﾝCV　空ﾊﾟﾚ排出完了
      LD      M596  ; 緩め部　ﾘｰﾀﾝCV押出ﾌﾟｯｼｬｰ後退
      LD      M419  ; 初期SOL励磁
      AND     M239  ; 緩め部　ﾘﾀｰﾝCV　押出ﾌﾟｯｼｬｰ後退端
      ORB
      ANI     M595  ; 緩め部　ﾘｰﾀﾝCV押出ﾌﾟｯｼｬｰ前進
      ORB
      AND     M17  ; 運転ﾓｰﾄﾞ切替
      AND     X0  ; 運転準備入り
      OUT     M596  ; 緩め部　ﾘｰﾀﾝCV押出ﾌﾟｯｼｬｰ後退
3281  LD      M595  ; 緩め部　ﾘｰﾀﾝCV押出ﾌﾟｯｼｬｰ前進
      ANI     Y303  ; 緩め部　ﾘﾀｰﾝCV　押出ﾌﾟｯｼｬ後退SOL
      OUT     Y302  ; 緩め部　ﾘﾀｰﾝCV　押出ﾌﾟｯｼｬ前進SOL
3284  LD      M596  ; 緩め部　ﾘｰﾀﾝCV押出ﾌﾟｯｼｬｰ後退
      ANI     Y302  ; 緩め部　ﾘﾀｰﾝCV　押出ﾌﾟｯｼｬ前進SOL
      OUT     Y303  ; 緩め部　ﾘﾀｰﾝCV　押出ﾌﾟｯｼｬ後退SOL
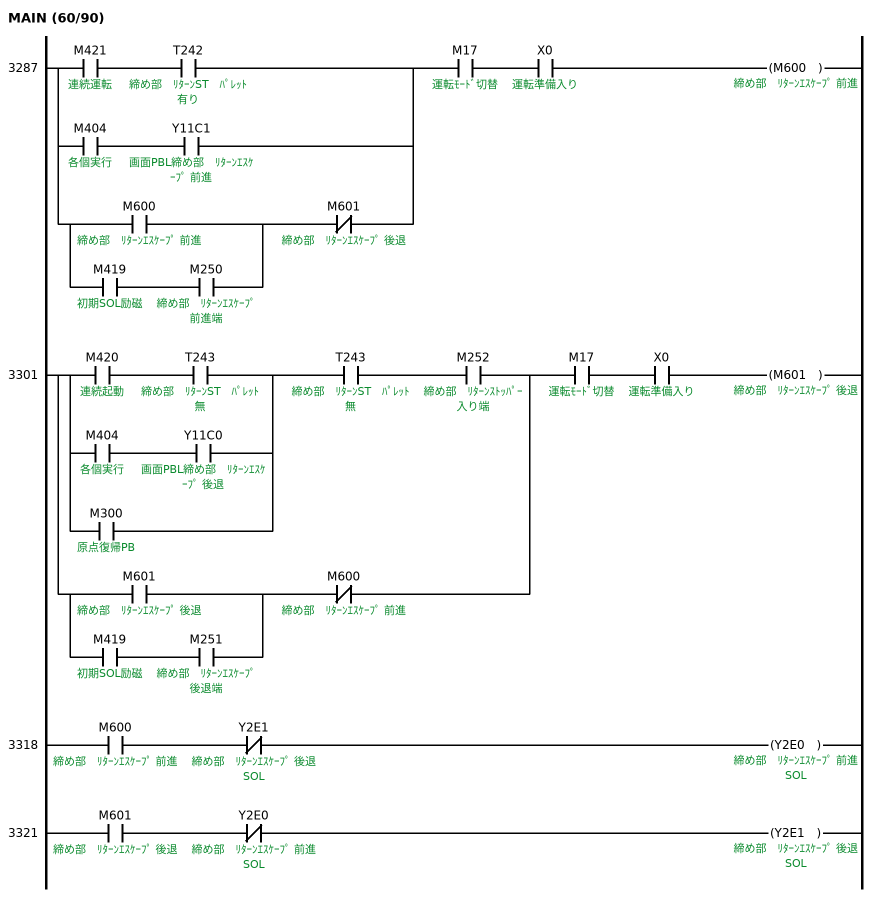
3287  LD      M421  ; 連続運転
      AND     T242  ; 締め部　ﾘﾀｰﾝST　ﾊﾟﾚｯﾄ有り
      LD      M404  ; 各個実行
      AND     Y11C1  ; 画面PBL締め部　ﾘﾀｰﾝｴｽｹｰﾌﾟ 前進
      ORB
      LD      M600  ; 締め部　ﾘﾀｰﾝｴｽｹｰﾌﾟ 前進
      LD      M419  ; 初期SOL励磁
      AND     M250  ; 締め部　ﾘﾀｰﾝｴｽｹｰﾌﾟ 前進端
      ORB
      ANI     M601  ; 締め部　ﾘﾀｰﾝｴｽｹｰﾌﾟ 後退
      ORB
      AND     M17  ; 運転ﾓｰﾄﾞ切替
      AND     X0  ; 運転準備入り
      OUT     M600  ; 締め部　ﾘﾀｰﾝｴｽｹｰﾌﾟ 前進
3301  LD      M420  ; 連続起動
      AND     T243  ; 締め部　ﾘﾀｰﾝST　ﾊﾟﾚｯﾄ無
      LD      M404  ; 各個実行
      AND     Y11C0  ; 画面PBL締め部　ﾘﾀｰﾝｴｽｹｰﾌﾟ 後退
      ORB
      OR      M300  ; 原点復帰PB
      AND     T243  ; 締め部　ﾘﾀｰﾝST　ﾊﾟﾚｯﾄ無
      AND     M252  ; 締め部　ﾘﾀｰﾝｽﾄｯﾊﾟｰ 入り端
      LD      M601  ; 締め部　ﾘﾀｰﾝｴｽｹｰﾌﾟ 後退
      LD      M419  ; 初期SOL励磁
      AND     M251  ; 締め部　ﾘﾀｰﾝｴｽｹｰﾌﾟ 後退端
      ORB
      ANI     M600  ; 締め部　ﾘﾀｰﾝｴｽｹｰﾌﾟ 前進
      ORB
      AND     M17  ; 運転ﾓｰﾄﾞ切替
      AND     X0  ; 運転準備入り
      OUT     M601  ; 締め部　ﾘﾀｰﾝｴｽｹｰﾌﾟ 後退
3318  LD      M600  ; 締め部　ﾘﾀｰﾝｴｽｹｰﾌﾟ 前進
      ANI     Y2E1  ; 締め部　ﾘﾀｰﾝｴｽｹｰﾌﾟ 後退 SOL
      OUT     Y2E0  ; 締め部　ﾘﾀｰﾝｴｽｹｰﾌﾟ 前進 SOL
3321  LD      M601  ; 締め部　ﾘﾀｰﾝｴｽｹｰﾌﾟ 後退
      ANI     Y2E0  ; 締め部　ﾘﾀｰﾝｴｽｹｰﾌﾟ 前進 SOL
      OUT     Y2E1  ; 締め部　ﾘﾀｰﾝｴｽｹｰﾌﾟ 後退 SOL
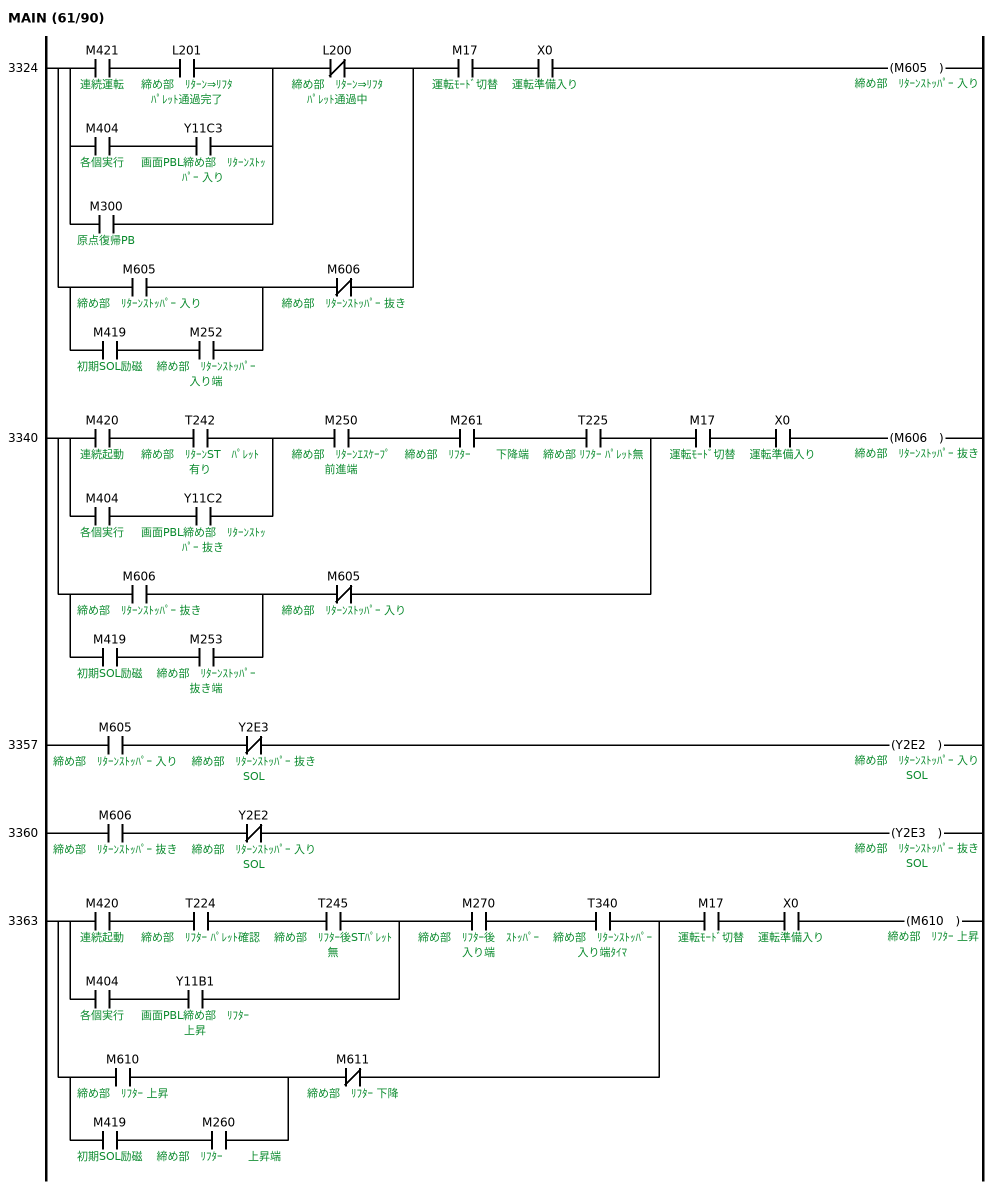
3324  LD      M421  ; 連続運転
      AND     L201  ; 締め部　ﾘﾀｰﾝ⇒ﾘﾌﾀ ﾊﾟﾚｯﾄ通過完了
      LD      M404  ; 各個実行
      AND     Y11C3  ; 画面PBL締め部　ﾘﾀｰﾝｽﾄｯﾊﾟｰ 入り
      ORB
      OR      M300  ; 原点復帰PB
      ANI     L200  ; 締め部　ﾘﾀｰﾝ⇒ﾘﾌﾀ ﾊﾟﾚｯﾄ通過中
      LD      M605  ; 締め部　ﾘﾀｰﾝｽﾄｯﾊﾟｰ 入り
      LD      M419  ; 初期SOL励磁
      AND     M252  ; 締め部　ﾘﾀｰﾝｽﾄｯﾊﾟｰ 入り端
      ORB
      ANI     M606  ; 締め部　ﾘﾀｰﾝｽﾄｯﾊﾟｰ 抜き
      ORB
      AND     M17  ; 運転ﾓｰﾄﾞ切替
      AND     X0  ; 運転準備入り
      OUT     M605  ; 締め部　ﾘﾀｰﾝｽﾄｯﾊﾟｰ 入り
3340  LD      M420  ; 連続起動
      AND     T242  ; 締め部　ﾘﾀｰﾝST　ﾊﾟﾚｯﾄ有り
      LD      M404  ; 各個実行
      AND     Y11C2  ; 画面PBL締め部　ﾘﾀｰﾝｽﾄｯﾊﾟｰ 抜き
      ORB
      AND     M250  ; 締め部　ﾘﾀｰﾝｴｽｹｰﾌﾟ 前進端
      AND     M261  ; 締め部　ﾘﾌﾀｰ 　　下降端
      AND     T225  ; 締め部 ﾘﾌﾀｰ ﾊﾟﾚｯﾄ無
      LD      M606  ; 締め部　ﾘﾀｰﾝｽﾄｯﾊﾟｰ 抜き
      LD      M419  ; 初期SOL励磁
      AND     M253  ; 締め部　ﾘﾀｰﾝｽﾄｯﾊﾟｰ 抜き端
      ORB
      ANI     M605  ; 締め部　ﾘﾀｰﾝｽﾄｯﾊﾟｰ 入り
      ORB
      AND     M17  ; 運転ﾓｰﾄﾞ切替
      AND     X0  ; 運転準備入り
      OUT     M606  ; 締め部　ﾘﾀｰﾝｽﾄｯﾊﾟｰ 抜き
3357  LD      M605  ; 締め部　ﾘﾀｰﾝｽﾄｯﾊﾟｰ 入り
      ANI     Y2E3  ; 締め部　ﾘﾀｰﾝｽﾄｯﾊﾟｰ 抜き SOL
      OUT     Y2E2  ; 締め部　ﾘﾀｰﾝｽﾄｯﾊﾟｰ 入り SOL
3360  LD      M606  ; 締め部　ﾘﾀｰﾝｽﾄｯﾊﾟｰ 抜き
      ANI     Y2E2  ; 締め部　ﾘﾀｰﾝｽﾄｯﾊﾟｰ 入り SOL
      OUT     Y2E3  ; 締め部　ﾘﾀｰﾝｽﾄｯﾊﾟｰ 抜き SOL
3363  LD      M420  ; 連続起動
      AND     T224  ; 締め部　ﾘﾌﾀｰ ﾊﾟﾚｯﾄ確認
      AND     T245  ; 締め部　ﾘﾌﾀｰ後STﾊﾟﾚｯﾄ無
      LD      M404  ; 各個実行
      AND     Y11B1  ; 画面PBL締め部　ﾘﾌﾀｰ 上昇
      ORB
      AND     M270  ; 締め部　ﾘﾌﾀｰ後　ｽﾄｯﾊﾟｰ　入り端
      AND     T340  ; 締め部　ﾘﾀｰﾝｽﾄｯﾊﾟｰ 入り端ﾀｲﾏ
      LD      M610  ; 締め部　ﾘﾌﾀｰ 上昇
      LD      M419  ; 初期SOL励磁
      AND     M260  ; 締め部　ﾘﾌﾀｰ 　　上昇端
      ORB
      ANI     M611  ; 締め部　ﾘﾌﾀｰ 下降
      ORB
      AND     M17  ; 運転ﾓｰﾄﾞ切替
      AND     X0  ; 運転準備入り
      OUT     M610  ; 締め部　ﾘﾌﾀｰ 上昇
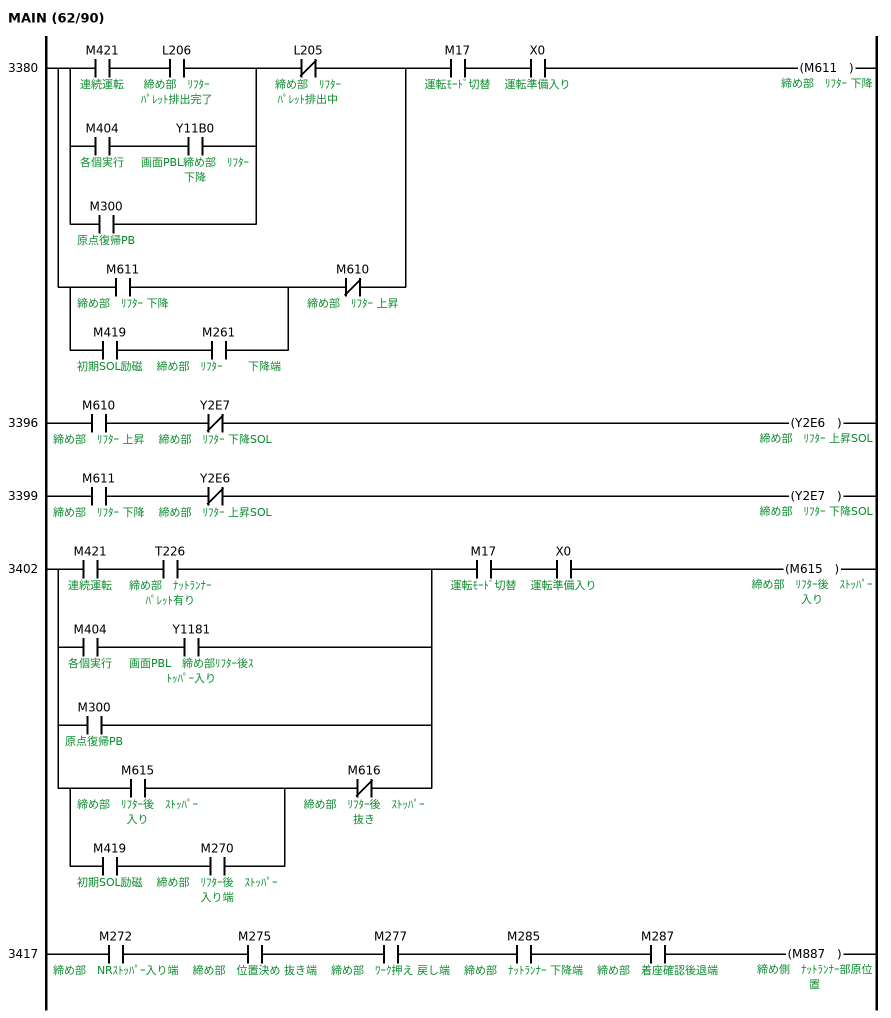
3380  LD      M421  ; 連続運転
      AND     L206  ; 締め部　ﾘﾌﾀｰ ﾊﾟﾚｯﾄ排出完了
      LD      M404  ; 各個実行
      AND     Y11B0  ; 画面PBL締め部　ﾘﾌﾀｰ 下降
      ORB
      OR      M300  ; 原点復帰PB
      ANI     L205  ; 締め部　ﾘﾌﾀｰ ﾊﾟﾚｯﾄ排出中
      LD      M611  ; 締め部　ﾘﾌﾀｰ 下降
      LD      M419  ; 初期SOL励磁
      AND     M261  ; 締め部　ﾘﾌﾀｰ 　　下降端
      ORB
      ANI     M610  ; 締め部　ﾘﾌﾀｰ 上昇
      ORB
      AND     M17  ; 運転ﾓｰﾄﾞ切替
      AND     X0  ; 運転準備入り
      OUT     M611  ; 締め部　ﾘﾌﾀｰ 下降
3396  LD      M610  ; 締め部　ﾘﾌﾀｰ 上昇
      ANI     Y2E7  ; 締め部　ﾘﾌﾀｰ 下降SOL
      OUT     Y2E6  ; 締め部　ﾘﾌﾀｰ 上昇SOL
3399  LD      M611  ; 締め部　ﾘﾌﾀｰ 下降
      ANI     Y2E6  ; 締め部　ﾘﾌﾀｰ 上昇SOL
      OUT     Y2E7  ; 締め部　ﾘﾌﾀｰ 下降SOL
3402  LD      M421  ; 連続運転
      AND     T226  ; 締め部　ﾅｯﾄﾗﾝﾅｰ ﾊﾟﾚｯﾄ有り
      LD      M404  ; 各個実行
      AND     Y1181  ; 画面PBL　締め部ﾘﾌﾀｰ後ｽﾄｯﾊﾟｰ入り
      ORB
      OR      M300  ; 原点復帰PB
      LD      M615  ; 締め部　ﾘﾌﾀｰ後　ｽﾄｯﾊﾟｰ　入り
      LD      M419  ; 初期SOL励磁
      AND     M270  ; 締め部　ﾘﾌﾀｰ後　ｽﾄｯﾊﾟｰ　入り端
      ORB
      ANI     M616  ; 締め部　ﾘﾌﾀｰ後　ｽﾄｯﾊﾟｰ　抜き
      ORB
      AND     M17  ; 運転ﾓｰﾄﾞ切替
      AND     X0  ; 運転準備入り
      OUT     M615  ; 締め部　ﾘﾌﾀｰ後　ｽﾄｯﾊﾟｰ　入り
3417  LD      M272  ; 締め部　NRｽﾄｯﾊﾟｰ入り端
      AND     M275  ; 締め部　位置決め 抜き端
      AND     M277  ; 締め部　ﾜｰｸ押え 戻し端
      AND     M285  ; 締め部　ﾅｯﾄﾗﾝﾅｰ 下降端
      AND     M287  ; 締め部　着座確認後退端
      OUT     M887  ; 締め側　ﾅｯﾄﾗﾝﾅｰ部原位置
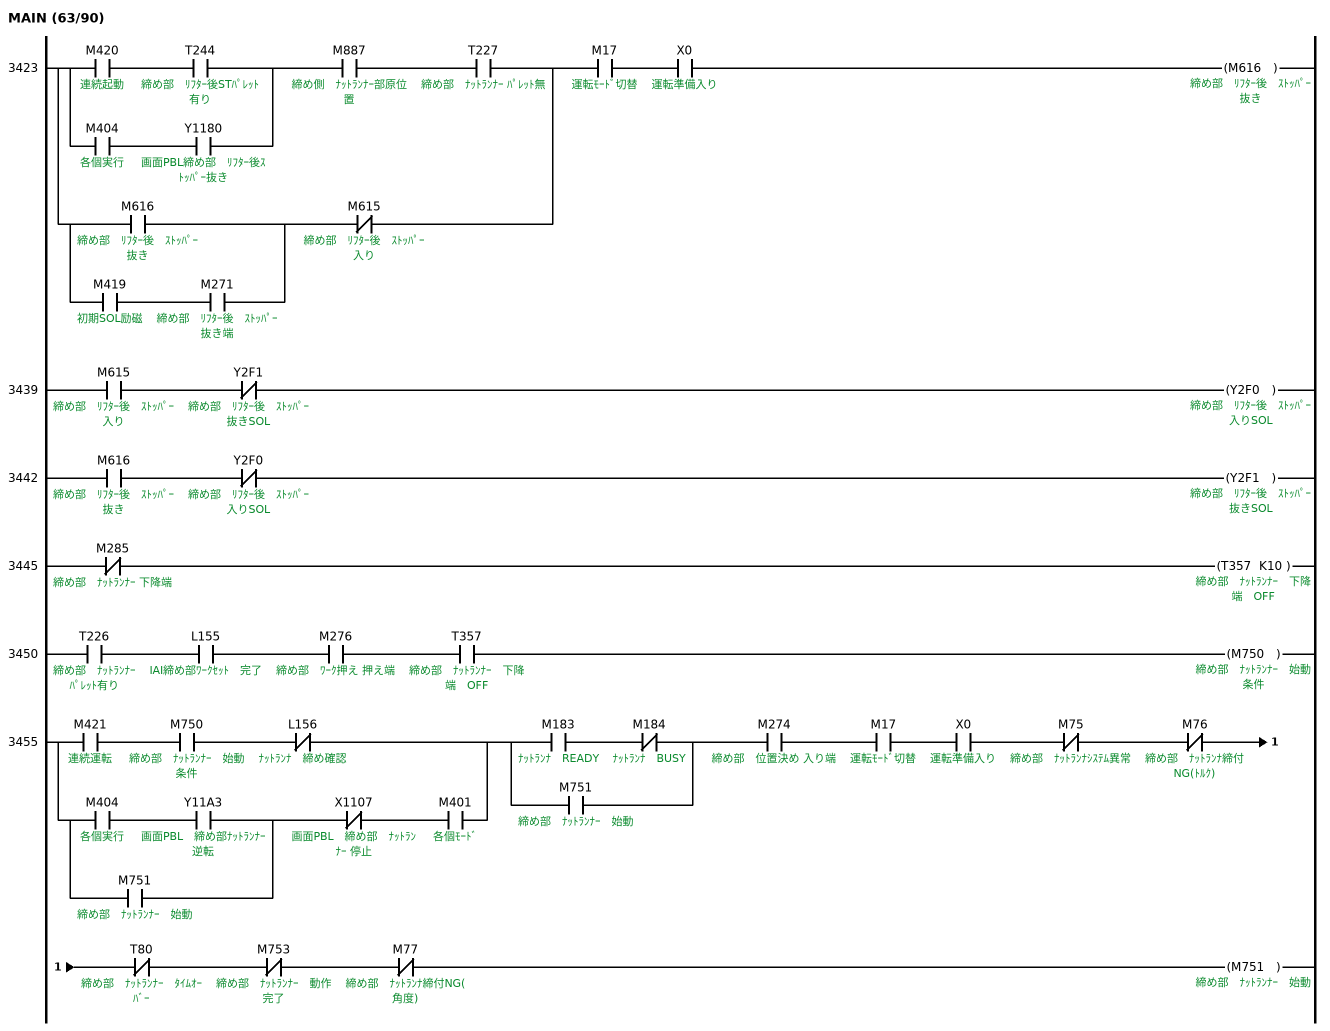
3423  LD      M420  ; 連続起動
      AND     T244  ; 締め部　ﾘﾌﾀｰ後STﾊﾟﾚｯﾄ有り
      LD      M404  ; 各個実行
      AND     Y1180  ; 画面PBL締め部　ﾘﾌﾀｰ後ｽﾄｯﾊﾟｰ抜き
      ORB
      AND     M887  ; 締め側　ﾅｯﾄﾗﾝﾅｰ部原位置
      AND     T227  ; 締め部　ﾅｯﾄﾗﾝﾅｰ ﾊﾟﾚｯﾄ無
      LD      M616  ; 締め部　ﾘﾌﾀｰ後　ｽﾄｯﾊﾟｰ　抜き
      LD      M419  ; 初期SOL励磁
      AND     M271  ; 締め部　ﾘﾌﾀｰ後　ｽﾄｯﾊﾟｰ　抜き端
      ORB
      ANI     M615  ; 締め部　ﾘﾌﾀｰ後　ｽﾄｯﾊﾟｰ　入り
      ORB
      AND     M17  ; 運転ﾓｰﾄﾞ切替
      AND     X0  ; 運転準備入り
      OUT     M616  ; 締め部　ﾘﾌﾀｰ後　ｽﾄｯﾊﾟｰ　抜き
3439  LD      M615  ; 締め部　ﾘﾌﾀｰ後　ｽﾄｯﾊﾟｰ　入り
      ANI     Y2F1  ; 締め部　ﾘﾌﾀｰ後　ｽﾄｯﾊﾟｰ　抜きSOL
      OUT     Y2F0  ; 締め部　ﾘﾌﾀｰ後　ｽﾄｯﾊﾟｰ　入りSOL
3442  LD      M616  ; 締め部　ﾘﾌﾀｰ後　ｽﾄｯﾊﾟｰ　抜き
      ANI     Y2F0  ; 締め部　ﾘﾌﾀｰ後　ｽﾄｯﾊﾟｰ　入りSOL
      OUT     Y2F1  ; 締め部　ﾘﾌﾀｰ後　ｽﾄｯﾊﾟｰ　抜きSOL
3445  LDI     M285  ; 締め部　ﾅｯﾄﾗﾝﾅｰ 下降端
      OUT     T357 K10  ; 締め部　ﾅｯﾄﾗﾝﾅｰ　下降端　OFF
3450  LD      T226  ; 締め部　ﾅｯﾄﾗﾝﾅｰ ﾊﾟﾚｯﾄ有り
      AND     L155  ; IAI締め部ﾜｰｸｾｯﾄ　完了
      AND     M276  ; 締め部　ﾜｰｸ押え 押え端
      AND     T357  ; 締め部　ﾅｯﾄﾗﾝﾅｰ　下降端　OFF
      OUT     M750  ; 締め部　ﾅｯﾄﾗﾝﾅｰ　始動条件
3455  LD      M421  ; 連続運転
      AND     M750  ; 締め部　ﾅｯﾄﾗﾝﾅｰ　始動条件
      ANI     L156  ; ﾅｯﾄﾗﾝﾅ　締め確認
      LD      M404  ; 各個実行
      AND     Y11A3  ; 画面PBL　締め部ﾅｯﾄﾗﾝﾅｰ 逆転
      OR      M751  ; 締め部　ﾅｯﾄﾗﾝﾅｰ　始動
      ANI     X1107  ; 画面PBL　締め部　ﾅｯﾄﾗﾝﾅｰ 停止
      AND     M401  ; 各個ﾓｰﾄﾞ
      ORB
      LD      M183  ; ﾅｯﾄﾗﾝﾅ　READY
      ANI     M184  ; ﾅｯﾄﾗﾝﾅ　BUSY
      OR      M751  ; 締め部　ﾅｯﾄﾗﾝﾅｰ　始動
      ANB
      AND     M274  ; 締め部　位置決め 入り端
      AND     M17  ; 運転ﾓｰﾄﾞ切替
      AND     X0  ; 運転準備入り
      ANI     M75  ; 締め部　ﾅｯﾄﾗﾝﾅｼｽﾃﾑ異常
      ANI     M76  ; 締め部　ﾅｯﾄﾗﾝﾅ締付 NG(ﾄﾙｸ)
      ANI     T80  ; 締め部　ﾅｯﾄﾗﾝﾅｰ　ﾀｲﾑｵｰﾊﾞｰ
      ANI     M753  ; 締め部　ﾅｯﾄﾗﾝﾅｰ　動作完了
      ANI     M77  ; 締め部　ﾅｯﾄﾗﾝﾅ締付NG(角度)
      OUT     M751  ; 締め部　ﾅｯﾄﾗﾝﾅｰ　始動
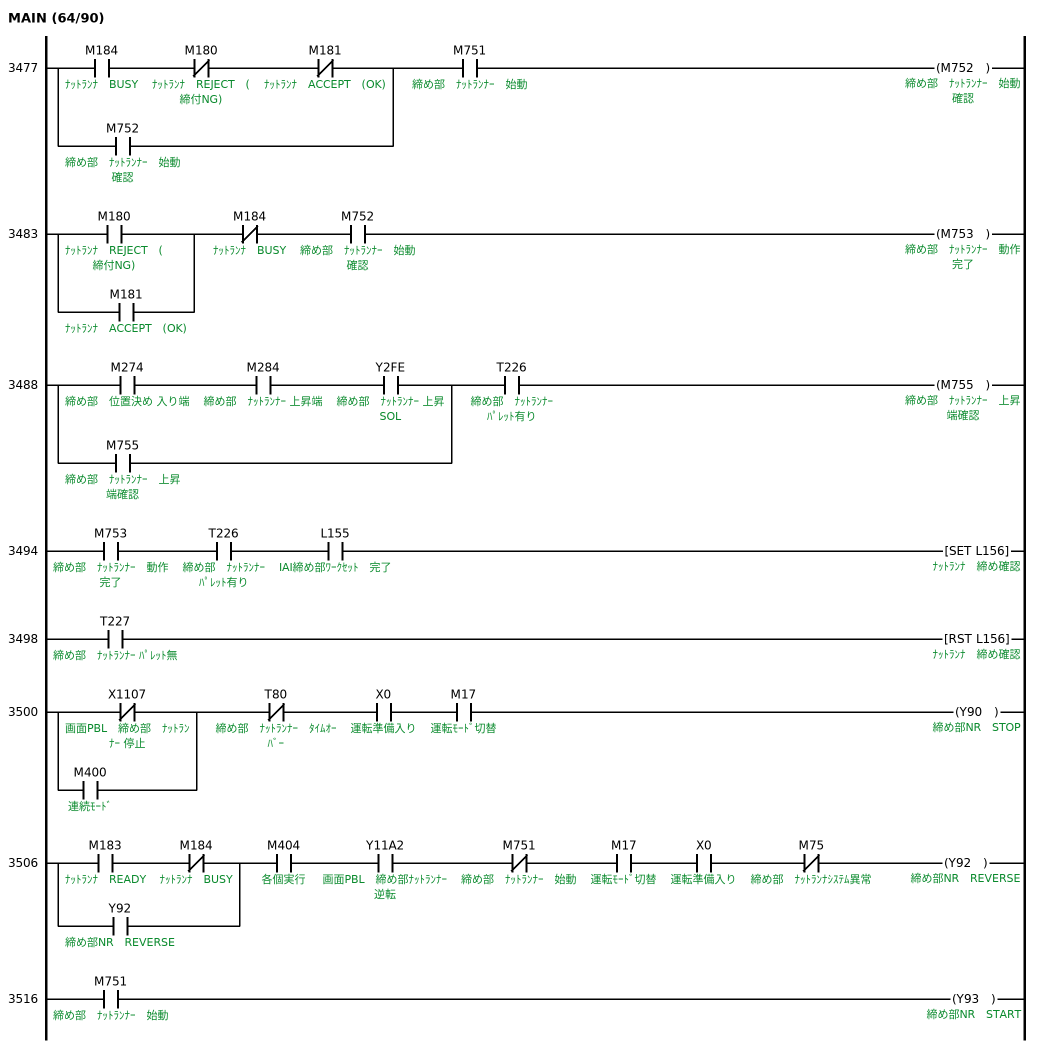
3477  LD      M184  ; ﾅｯﾄﾗﾝﾅ　BUSY
      ANI     M180  ; ﾅｯﾄﾗﾝﾅ　REJECT　(締付NG)
      ANI     M181  ; ﾅｯﾄﾗﾝﾅ　ACCEPT　(OK)
      OR      M752  ; 締め部　ﾅｯﾄﾗﾝﾅｰ　始動確認
      AND     M751  ; 締め部　ﾅｯﾄﾗﾝﾅｰ　始動
      OUT     M752  ; 締め部　ﾅｯﾄﾗﾝﾅｰ　始動確認
3483  LD      M180  ; ﾅｯﾄﾗﾝﾅ　REJECT　(締付NG)
      OR      M181  ; ﾅｯﾄﾗﾝﾅ　ACCEPT　(OK)
      ANI     M184  ; ﾅｯﾄﾗﾝﾅ　BUSY
      AND     M752  ; 締め部　ﾅｯﾄﾗﾝﾅｰ　始動確認
      OUT     M753  ; 締め部　ﾅｯﾄﾗﾝﾅｰ　動作完了
3488  LD      M274  ; 締め部　位置決め 入り端
      AND     M284  ; 締め部　ﾅｯﾄﾗﾝﾅｰ 上昇端
      AND     Y2FE  ; 締め部　ﾅｯﾄﾗﾝﾅｰ 上昇 SOL
      OR      M755  ; 締め部　ﾅｯﾄﾗﾝﾅｰ　上昇端確認
      AND     T226  ; 締め部　ﾅｯﾄﾗﾝﾅｰ ﾊﾟﾚｯﾄ有り
      OUT     M755  ; 締め部　ﾅｯﾄﾗﾝﾅｰ　上昇端確認
3494  LD      M753  ; 締め部　ﾅｯﾄﾗﾝﾅｰ　動作完了
      AND     T226  ; 締め部　ﾅｯﾄﾗﾝﾅｰ ﾊﾟﾚｯﾄ有り
      AND     L155  ; IAI締め部ﾜｰｸｾｯﾄ　完了
      SET     L156  ; ﾅｯﾄﾗﾝﾅ　締め確認
3498  LD      T227  ; 締め部　ﾅｯﾄﾗﾝﾅｰ ﾊﾟﾚｯﾄ無
      RST     L156  ; ﾅｯﾄﾗﾝﾅ　締め確認
3500  LDI     X1107  ; 画面PBL　締め部　ﾅｯﾄﾗﾝﾅｰ 停止
      OR      M400  ; 連続ﾓｰﾄﾞ
      ANI     T80  ; 締め部　ﾅｯﾄﾗﾝﾅｰ　ﾀｲﾑｵｰﾊﾞｰ
      AND     X0  ; 運転準備入り
      AND     M17  ; 運転ﾓｰﾄﾞ切替
      OUT     Y90  ; 締め部NR　STOP
3506  LD      M183  ; ﾅｯﾄﾗﾝﾅ　READY
      ANI     M184  ; ﾅｯﾄﾗﾝﾅ　BUSY
      OR      Y92  ; 締め部NR　REVERSE
      AND     M404  ; 各個実行
      AND     Y11A2  ; 画面PBL　締め部ﾅｯﾄﾗﾝﾅｰ 逆転
      ANI     M751  ; 締め部　ﾅｯﾄﾗﾝﾅｰ　始動
      AND     M17  ; 運転ﾓｰﾄﾞ切替
      AND     X0  ; 運転準備入り
      ANI     M75  ; 締め部　ﾅｯﾄﾗﾝﾅｼｽﾃﾑ異常
      OUT     Y92  ; 締め部NR　REVERSE
3516  LD      M751  ; 締め部　ﾅｯﾄﾗﾝﾅｰ　始動
      OUT     Y93  ; 締め部NR　START
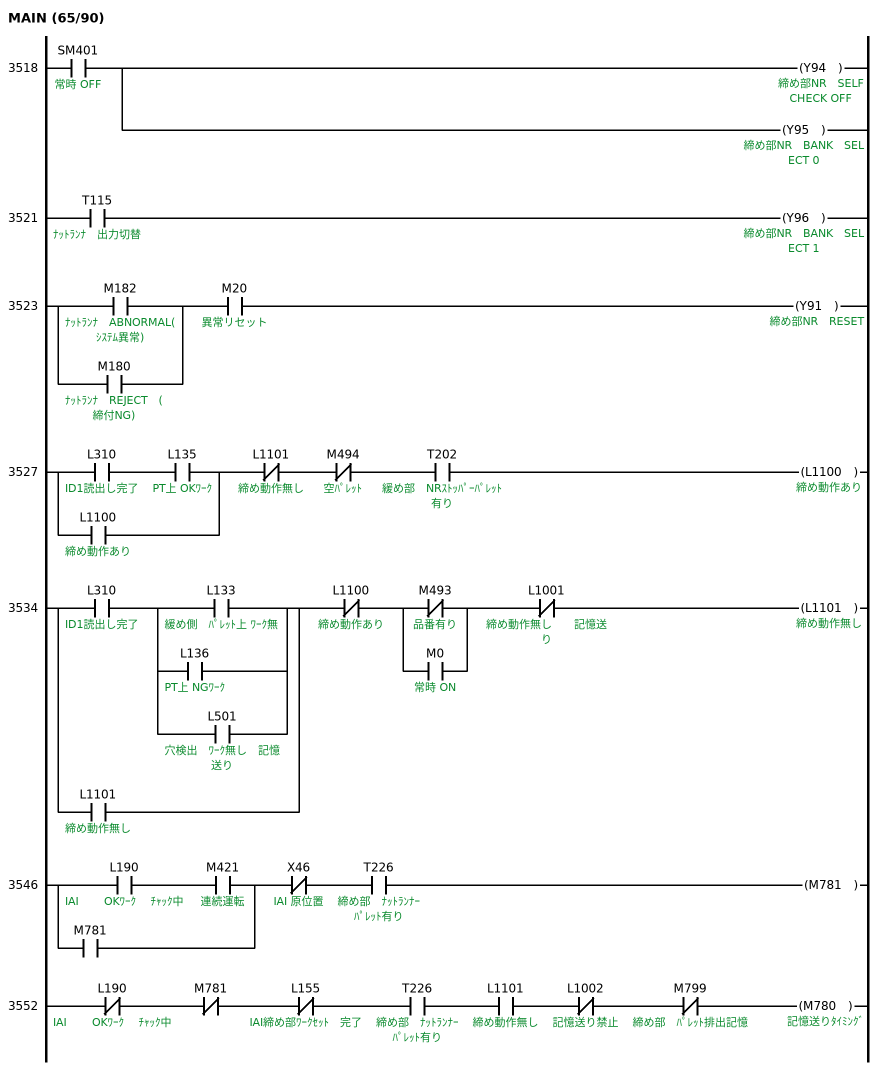
3518  LD      SM401  ; 常時 OFF
      OUT     Y94  ; 締め部NR　SELF CHECK OFF
      OUT     Y95  ; 締め部NR　BANK　SELECT 0
3521  LD      T115  ; ﾅｯﾄﾗﾝﾅ　出力切替
      OUT     Y96  ; 締め部NR　BANK　SELECT 1
3523  LD      M182  ; ﾅｯﾄﾗﾝﾅ　ABNORMAL(ｼｽﾃﾑ異常)
      OR      M180  ; ﾅｯﾄﾗﾝﾅ　REJECT　(締付NG)
      AND     M20  ; 異常リセット
      OUT     Y91  ; 締め部NR　RESET
3527  LD      L310  ; ID1読出し完了
      AND     L135  ; PT上 OKﾜｰｸ
      OR      L1100  ; 締め動作あり
      ANI     L1101  ; 締め動作無し
      ANI     M494  ; 空ﾊﾟﾚｯﾄ
      AND     T202  ; 緩め部　NRｽﾄｯﾊﾟｰﾊﾟﾚｯﾄ有り
      OUT     L1100  ; 締め動作あり
3534  LD      L310  ; ID1読出し完了
      LD      L133  ; 緩め側　ﾊﾟﾚｯﾄ上 ﾜｰｸ無
      OR      L136  ; PT上 NGﾜｰｸ
      OR      L501  ; 穴検出　ﾜｰｸ無し　記憶送り
      ANB
      OR      L1101  ; 締め動作無し
      ANI     L1100  ; 締め動作あり
      LDI     M493  ; 品番有り
      OR      M0  ; 常時 ON
      ANB
      ANI     L1001  ; 締め動作無し　　記憶送り
      OUT     L1101  ; 締め動作無し
3546  LD      L190  ; IAI　　 OKﾜｰｸ　 ﾁｬｯｸ中
      AND     M421  ; 連続運転
      OR      M781
      ANI     X46  ; IAI 原位置
      AND     T226  ; 締め部　ﾅｯﾄﾗﾝﾅｰ ﾊﾟﾚｯﾄ有り
      OUT     M781
3552  LDI     L190  ; IAI　　 OKﾜｰｸ　 ﾁｬｯｸ中
      ANI     M781
      ANI     L155  ; IAI締め部ﾜｰｸｾｯﾄ　完了
      AND     T226  ; 締め部　ﾅｯﾄﾗﾝﾅｰ ﾊﾟﾚｯﾄ有り
      AND     L1101  ; 締め動作無し
      ANI     L1002  ; 記憶送り禁止
      ANI     M799  ; 締め部　ﾊﾟﾚｯﾄ排出記憶
      OUT     M780  ; 記憶送りﾀｲﾐﾝｸﾞ
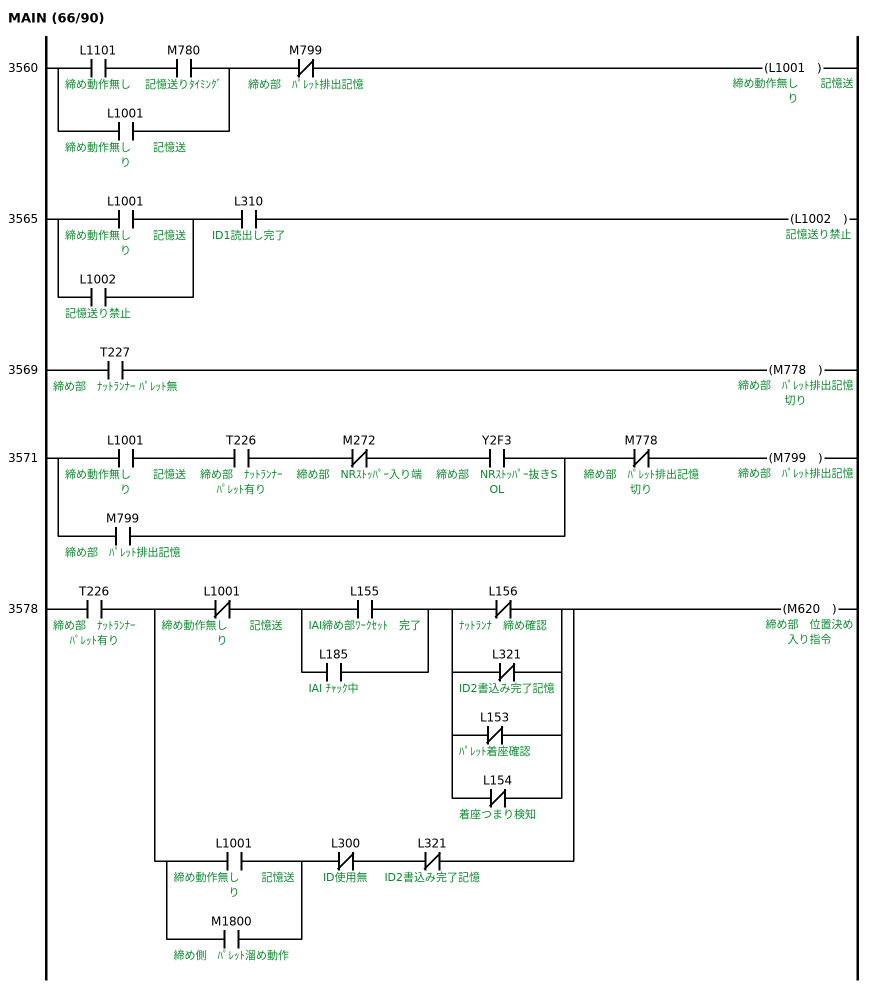
3560  LD      L1101  ; 締め動作無し
      AND     M780  ; 記憶送りﾀｲﾐﾝｸﾞ
      OR      L1001  ; 締め動作無し　　記憶送り
      ANI     M799  ; 締め部　ﾊﾟﾚｯﾄ排出記憶
      OUT     L1001  ; 締め動作無し　　記憶送り
3565  LD      L1001  ; 締め動作無し　　記憶送り
      OR      L1002  ; 記憶送り禁止
      AND     L310  ; ID1読出し完了
      OUT     L1002  ; 記憶送り禁止
3569  LD      T227  ; 締め部　ﾅｯﾄﾗﾝﾅｰ ﾊﾟﾚｯﾄ無
      OUT     M778  ; 締め部　ﾊﾟﾚｯﾄ排出記憶切り
3571  LD      L1001  ; 締め動作無し　　記憶送り
      AND     T226  ; 締め部　ﾅｯﾄﾗﾝﾅｰ ﾊﾟﾚｯﾄ有り
      ANI     M272  ; 締め部　NRｽﾄｯﾊﾟｰ入り端
      AND     Y2F3  ; 締め部　NRｽﾄｯﾊﾟｰ抜きSOL
      OR      M799  ; 締め部　ﾊﾟﾚｯﾄ排出記憶
      ANI     M778  ; 締め部　ﾊﾟﾚｯﾄ排出記憶切り
      OUT     M799  ; 締め部　ﾊﾟﾚｯﾄ排出記憶
3578  LD      T226  ; 締め部　ﾅｯﾄﾗﾝﾅｰ ﾊﾟﾚｯﾄ有り
      LDI     L1001  ; 締め動作無し　　記憶送り
      LD      L155  ; IAI締め部ﾜｰｸｾｯﾄ　完了
      OR      L185  ; IAI ﾁｬｯｸ中
      ANB
      LDI     L156  ; ﾅｯﾄﾗﾝﾅ　締め確認
      ORI     L321  ; ID2書込み完了記憶
      ORI     L153  ; ﾊﾟﾚｯﾄ着座確認
      ORI     L154  ; 着座つまり検知
      ANB
      LD      L1001  ; 締め動作無し　　記憶送り
      OR      M1800  ; 締め側　ﾊﾟﾚｯﾄ溜め動作
      ANI     L300  ; ID使用無
      ANI     L321  ; ID2書込み完了記憶
      ORB
      ANB
      OUT     M620  ; 締め部　位置決め 入り指令
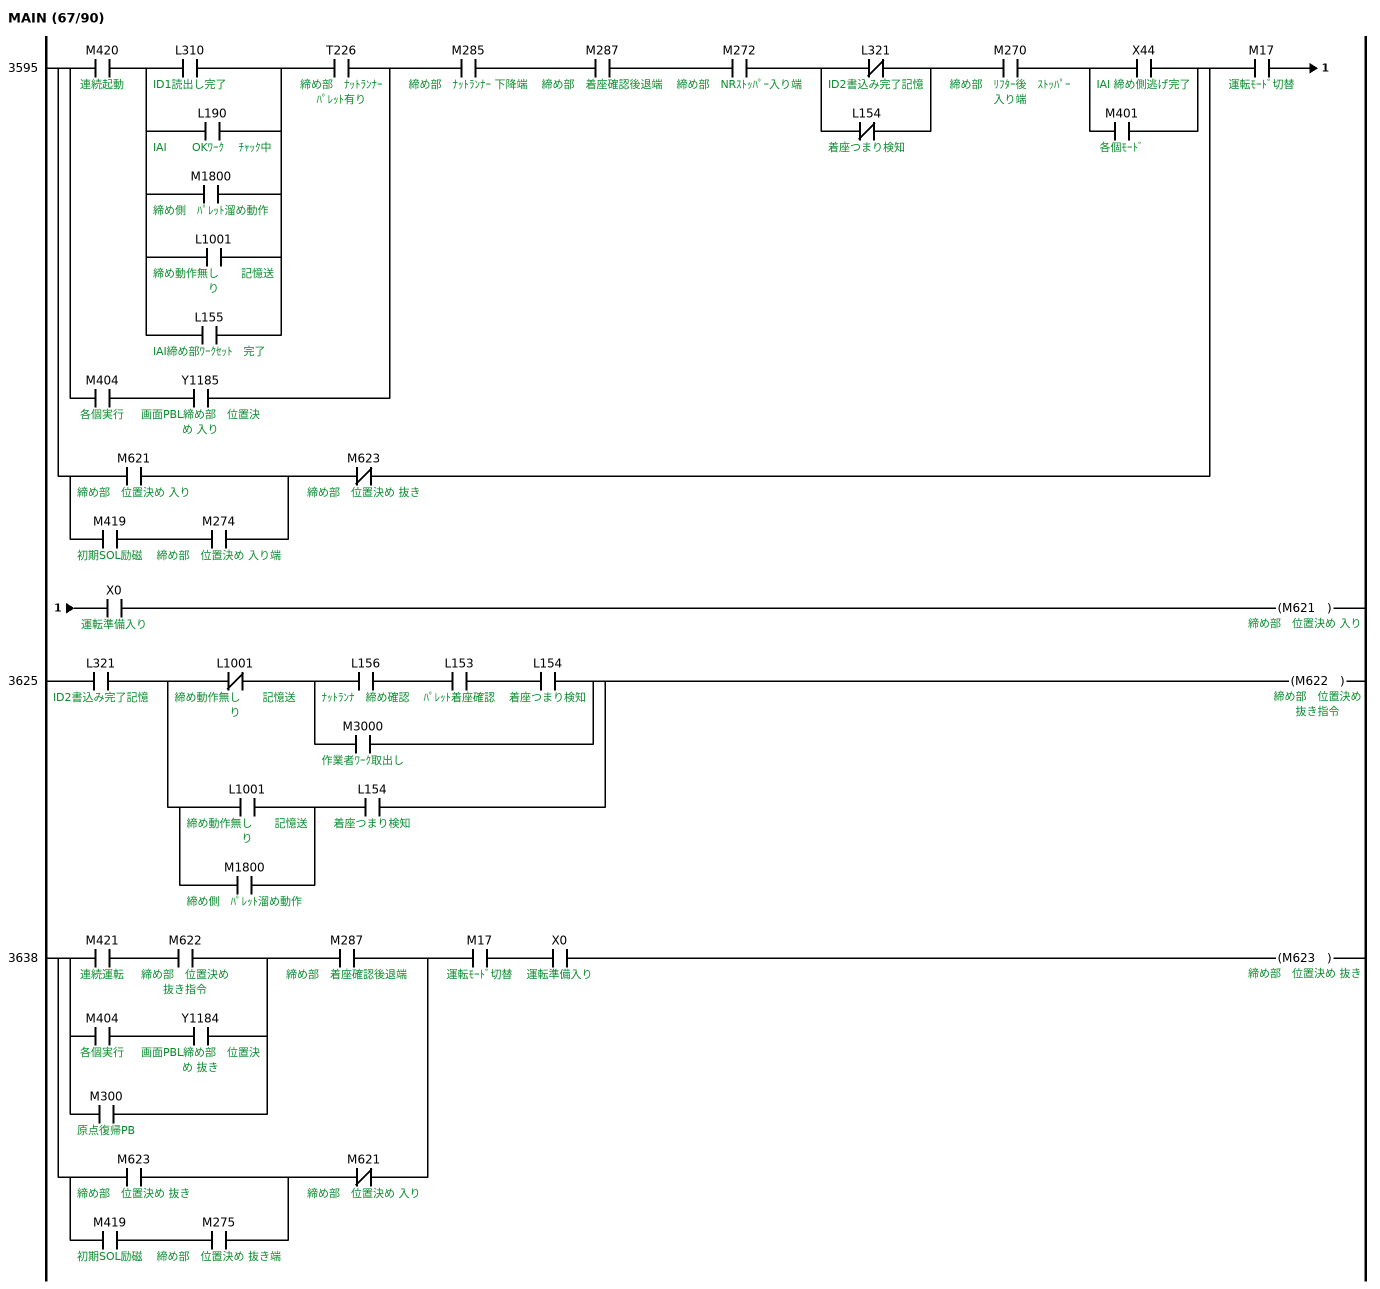
3595  LD      M420  ; 連続起動
      LD      L310  ; ID1読出し完了
      OR      L190  ; IAI　　 OKﾜｰｸ　 ﾁｬｯｸ中
      OR      M1800  ; 締め側　ﾊﾟﾚｯﾄ溜め動作
      OR      L1001  ; 締め動作無し　　記憶送り
      OR      L155  ; IAI締め部ﾜｰｸｾｯﾄ　完了
      ANB
      AND     T226  ; 締め部　ﾅｯﾄﾗﾝﾅｰ ﾊﾟﾚｯﾄ有り
      LD      M404  ; 各個実行
      AND     Y1185  ; 画面PBL締め部　位置決め 入り
      ORB
      AND     M285  ; 締め部　ﾅｯﾄﾗﾝﾅｰ 下降端
      AND     M287  ; 締め部　着座確認後退端
      AND     M272  ; 締め部　NRｽﾄｯﾊﾟｰ入り端
      LDI     L321  ; ID2書込み完了記憶
      ORI     L154  ; 着座つまり検知
      ANB
      AND     M270  ; 締め部　ﾘﾌﾀｰ後　ｽﾄｯﾊﾟｰ　入り端
      LD      X44  ; IAI 締め側逃げ完了
      OR      M401  ; 各個ﾓｰﾄﾞ
      ANB
      LD      M621  ; 締め部　位置決め 入り
      LD      M419  ; 初期SOL励磁
      AND     M274  ; 締め部　位置決め 入り端
      ORB
      ANI     M623  ; 締め部　位置決め 抜き
      ORB
      AND     M17  ; 運転ﾓｰﾄﾞ切替
      AND     X0  ; 運転準備入り
      OUT     M621  ; 締め部　位置決め 入り
3625  LD      L321  ; ID2書込み完了記憶
      LDI     L1001  ; 締め動作無し　　記憶送り
      LD      L156  ; ﾅｯﾄﾗﾝﾅ　締め確認
      AND     L153  ; ﾊﾟﾚｯﾄ着座確認
      AND     L154  ; 着座つまり検知
      OR      M3000  ; 作業者ﾜｰｸ取出し
      ANB
      LD      L1001  ; 締め動作無し　　記憶送り
      OR      M1800  ; 締め側　ﾊﾟﾚｯﾄ溜め動作
      AND     L154  ; 着座つまり検知
      ORB
      ANB
      OUT     M622  ; 締め部　位置決め 抜き指令
3638  LD      M421  ; 連続運転
      AND     M622  ; 締め部　位置決め 抜き指令
      LD      M404  ; 各個実行
      AND     Y1184  ; 画面PBL締め部　位置決め 抜き
      ORB
      OR      M300  ; 原点復帰PB
      AND     M287  ; 締め部　着座確認後退端
      LD      M623  ; 締め部　位置決め 抜き
      LD      M419  ; 初期SOL励磁
      AND     M275  ; 締め部　位置決め 抜き端
      ORB
      ANI     M621  ; 締め部　位置決め 入り
      ORB
      AND     M17  ; 運転ﾓｰﾄﾞ切替
      AND     X0  ; 運転準備入り
      OUT     M623  ; 締め部　位置決め 抜き
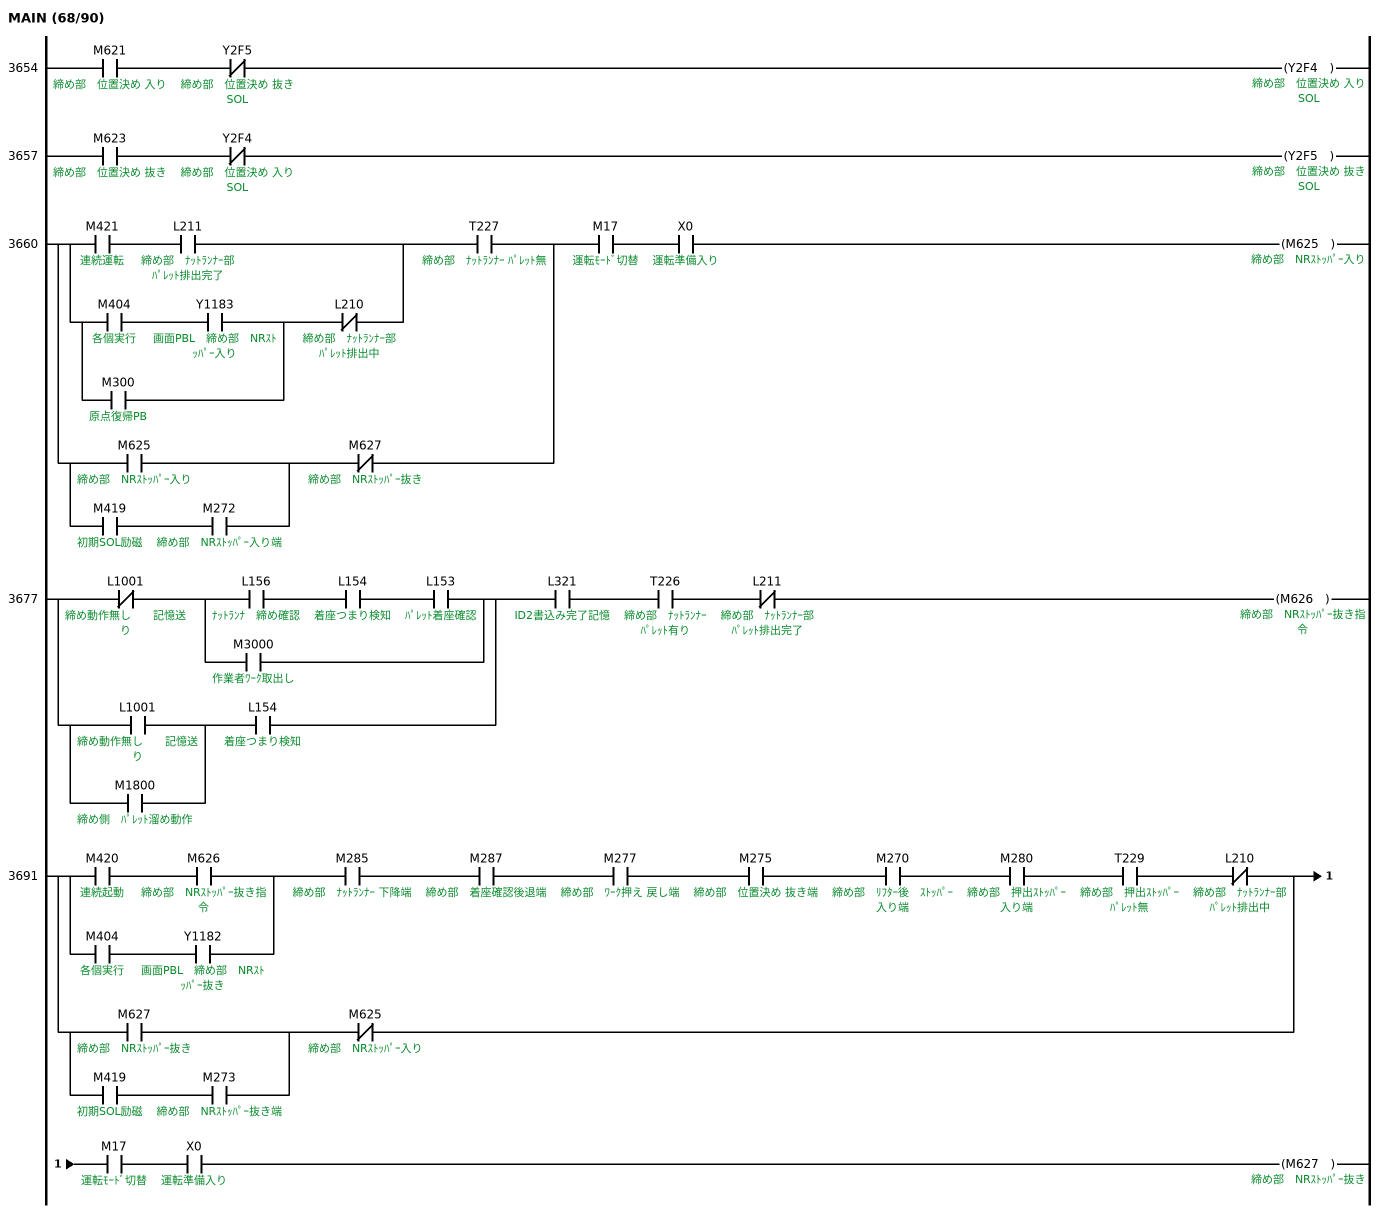
3654  LD      M621  ; 締め部　位置決め 入り
      ANI     Y2F5  ; 締め部　位置決め 抜き SOL
      OUT     Y2F4  ; 締め部　位置決め 入り SOL
3657  LD      M623  ; 締め部　位置決め 抜き
      ANI     Y2F4  ; 締め部　位置決め 入り SOL
      OUT     Y2F5  ; 締め部　位置決め 抜き SOL
3660  LD      M421  ; 連続運転
      AND     L211  ; 締め部　ﾅｯﾄﾗﾝﾅｰ部 ﾊﾟﾚｯﾄ排出完了
      LD      M404  ; 各個実行
      AND     Y1183  ; 画面PBL　締め部　NRｽﾄｯﾊﾟｰ入り
      OR      M300  ; 原点復帰PB
      ANI     L210  ; 締め部　ﾅｯﾄﾗﾝﾅｰ部 ﾊﾟﾚｯﾄ排出中
      ORB
      AND     T227  ; 締め部　ﾅｯﾄﾗﾝﾅｰ ﾊﾟﾚｯﾄ無
      LD      M625  ; 締め部　NRｽﾄｯﾊﾟｰ入り
      LD      M419  ; 初期SOL励磁
      AND     M272  ; 締め部　NRｽﾄｯﾊﾟｰ入り端
      ORB
      ANI     M627  ; 締め部　NRｽﾄｯﾊﾟｰ抜き
      ORB
      AND     M17  ; 運転ﾓｰﾄﾞ切替
      AND     X0  ; 運転準備入り
      OUT     M625  ; 締め部　NRｽﾄｯﾊﾟｰ入り
3677  LDI     L1001  ; 締め動作無し　　記憶送り
      LD      L156  ; ﾅｯﾄﾗﾝﾅ　締め確認
      AND     L154  ; 着座つまり検知
      AND     L153  ; ﾊﾟﾚｯﾄ着座確認
      OR      M3000  ; 作業者ﾜｰｸ取出し
      ANB
      LD      L1001  ; 締め動作無し　　記憶送り
      OR      M1800  ; 締め側　ﾊﾟﾚｯﾄ溜め動作
      AND     L154  ; 着座つまり検知
      ORB
      AND     L321  ; ID2書込み完了記憶
      AND     T226  ; 締め部　ﾅｯﾄﾗﾝﾅｰ ﾊﾟﾚｯﾄ有り
      ANI     L211  ; 締め部　ﾅｯﾄﾗﾝﾅｰ部 ﾊﾟﾚｯﾄ排出完了
      OUT     M626  ; 締め部　NRｽﾄｯﾊﾟｰ抜き指令
3691  LD      M420  ; 連続起動
      AND     M626  ; 締め部　NRｽﾄｯﾊﾟｰ抜き指令
      LD      M404  ; 各個実行
      AND     Y1182  ; 画面PBL　締め部　NRｽﾄｯﾊﾟｰ抜き
      ORB
      AND     M285  ; 締め部　ﾅｯﾄﾗﾝﾅｰ 下降端
      AND     M287  ; 締め部　着座確認後退端
      AND     M277  ; 締め部　ﾜｰｸ押え 戻し端
      AND     M275  ; 締め部　位置決め 抜き端
      AND     M270  ; 締め部　ﾘﾌﾀｰ後　ｽﾄｯﾊﾟｰ　入り端
      AND     M280  ; 締め部　押出ｽﾄｯﾊﾟｰ 入り端
      AND     T229  ; 締め部　押出ｽﾄｯﾊﾟｰ ﾊﾟﾚｯﾄ無
      ANI     L210  ; 締め部　ﾅｯﾄﾗﾝﾅｰ部 ﾊﾟﾚｯﾄ排出中
      LD      M627  ; 締め部　NRｽﾄｯﾊﾟｰ抜き
      LD      M419  ; 初期SOL励磁
      AND     M273  ; 締め部　NRｽﾄｯﾊﾟｰ抜き端
      ORB
      ANI     M625  ; 締め部　NRｽﾄｯﾊﾟｰ入り
      ORB
      AND     M17  ; 運転ﾓｰﾄﾞ切替
      AND     X0  ; 運転準備入り
      OUT     M627  ; 締め部　NRｽﾄｯﾊﾟｰ抜き
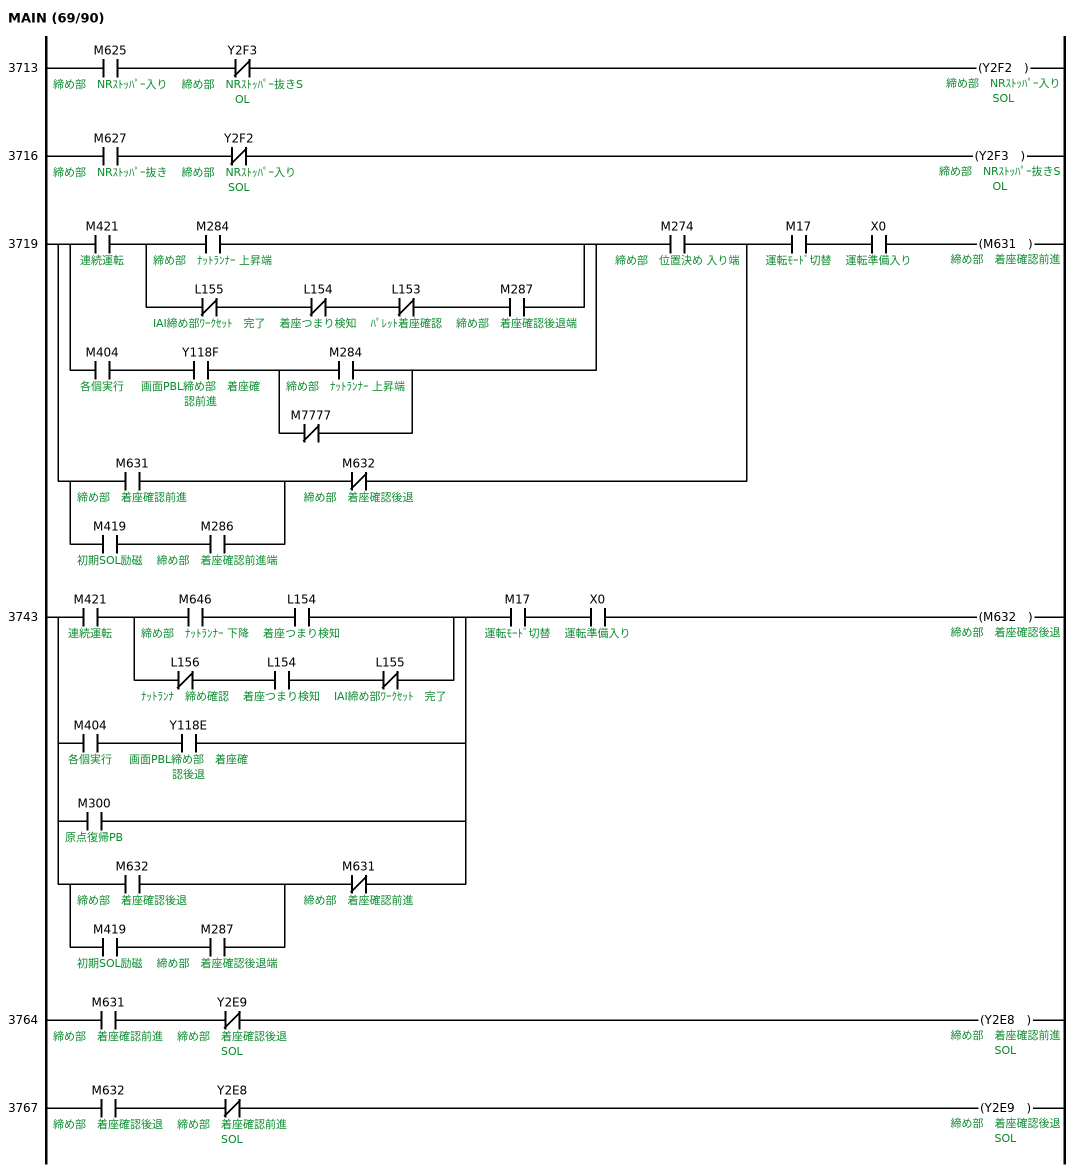
3713  LD      M625  ; 締め部　NRｽﾄｯﾊﾟｰ入り
      ANI     Y2F3  ; 締め部　NRｽﾄｯﾊﾟｰ抜きSOL
      OUT     Y2F2  ; 締め部　NRｽﾄｯﾊﾟｰ入り SOL
3716  LD      M627  ; 締め部　NRｽﾄｯﾊﾟｰ抜き
      ANI     Y2F2  ; 締め部　NRｽﾄｯﾊﾟｰ入り SOL
      OUT     Y2F3  ; 締め部　NRｽﾄｯﾊﾟｰ抜きSOL
3719  LD      M421  ; 連続運転
      LD      M284  ; 締め部　ﾅｯﾄﾗﾝﾅｰ 上昇端
      LDI     L155  ; IAI締め部ﾜｰｸｾｯﾄ　完了
      ANI     L154  ; 着座つまり検知
      ANI     L153  ; ﾊﾟﾚｯﾄ着座確認
      AND     M287  ; 締め部　着座確認後退端
      ORB
      ANB
      LD      M404  ; 各個実行
      AND     Y118F  ; 画面PBL締め部　着座確認前進
      LD      M284  ; 締め部　ﾅｯﾄﾗﾝﾅｰ 上昇端
      ORI     M7777
      ANB
      ORB
      AND     M274  ; 締め部　位置決め 入り端
      LD      M631  ; 締め部　着座確認前進
      LD      M419  ; 初期SOL励磁
      AND     M286  ; 締め部　着座確認前進端
      ORB
      ANI     M632  ; 締め部　着座確認後退
      ORB
      AND     M17  ; 運転ﾓｰﾄﾞ切替
      AND     X0  ; 運転準備入り
      OUT     M631  ; 締め部　着座確認前進
3743  LD      M421  ; 連続運転
      LD      M646  ; 締め部　ﾅｯﾄﾗﾝﾅｰ 下降
      AND     L154  ; 着座つまり検知
      LDI     L156  ; ﾅｯﾄﾗﾝﾅ　締め確認
      AND     L154  ; 着座つまり検知
      ANI     L155  ; IAI締め部ﾜｰｸｾｯﾄ　完了
      ORB
      ANB
      LD      M404  ; 各個実行
      AND     Y118E  ; 画面PBL締め部　着座確認後退
      ORB
      OR      M300  ; 原点復帰PB
      LD      M632  ; 締め部　着座確認後退
      LD      M419  ; 初期SOL励磁
      AND     M287  ; 締め部　着座確認後退端
      ORB
      ANI     M631  ; 締め部　着座確認前進
      ORB
      AND     M17  ; 運転ﾓｰﾄﾞ切替
      AND     X0  ; 運転準備入り
      OUT     M632  ; 締め部　着座確認後退
3764  LD      M631  ; 締め部　着座確認前進
      ANI     Y2E9  ; 締め部　着座確認後退 SOL
      OUT     Y2E8  ; 締め部　着座確認前進 SOL
3767  LD      M632  ; 締め部　着座確認後退
      ANI     Y2E8  ; 締め部　着座確認前進 SOL
      OUT     Y2E9  ; 締め部　着座確認後退 SOL
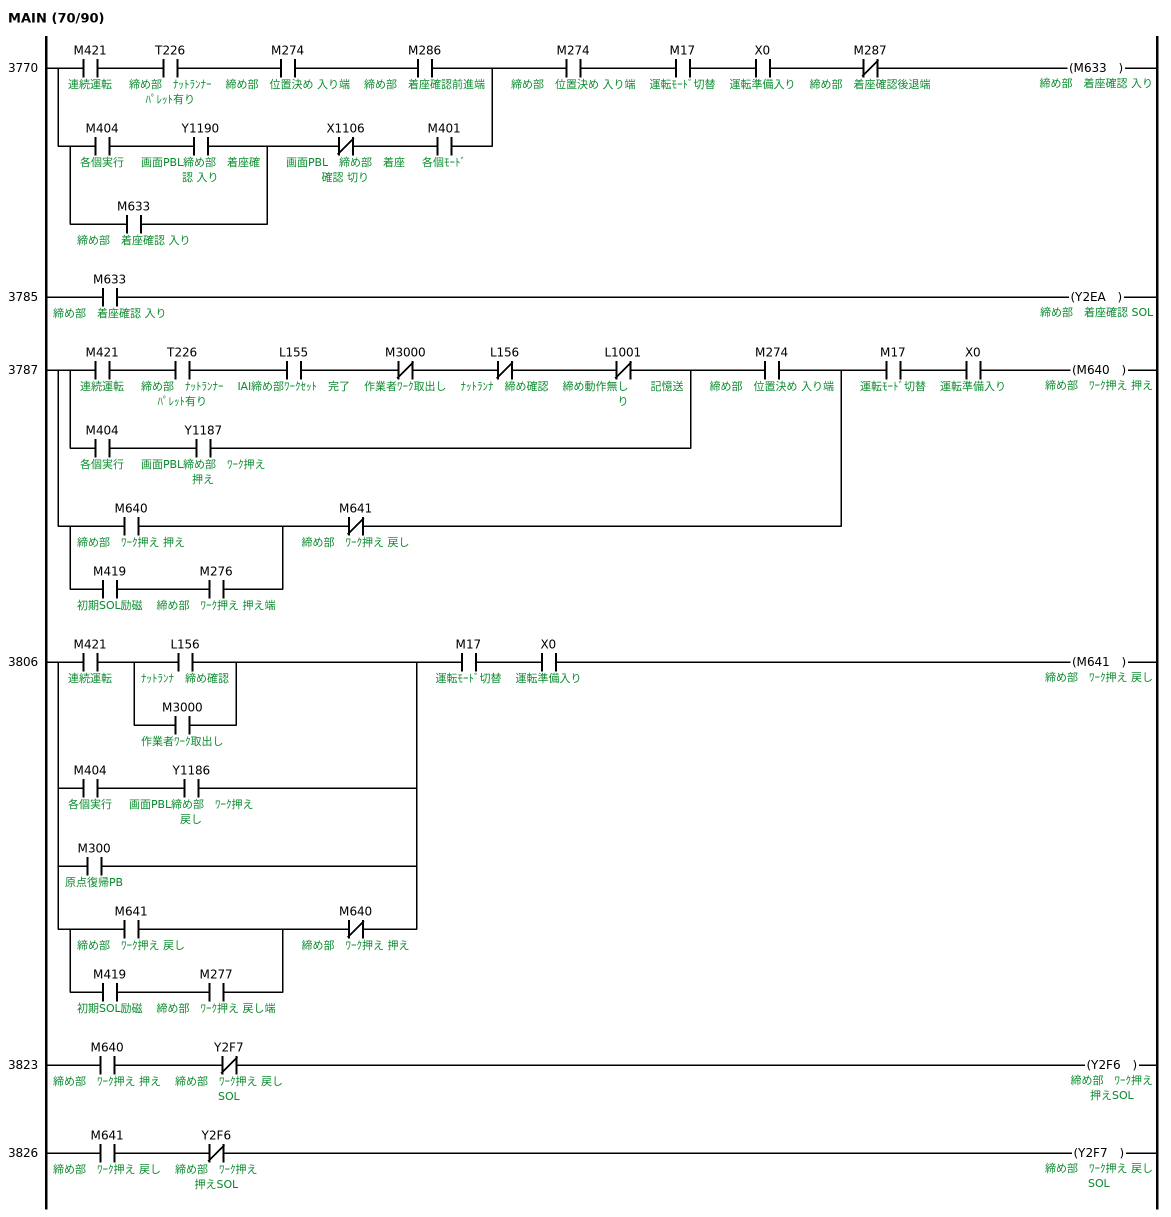
3770  LD      M421  ; 連続運転
      AND     T226  ; 締め部　ﾅｯﾄﾗﾝﾅｰ ﾊﾟﾚｯﾄ有り
      AND     M274  ; 締め部　位置決め 入り端
      AND     M286  ; 締め部　着座確認前進端
      LD      M404  ; 各個実行
      AND     Y1190  ; 画面PBL締め部　着座確認 入り
      OR      M633  ; 締め部　着座確認 入り
      ANI     X1106  ; 画面PBL　締め部　着座確認 切り
      AND     M401  ; 各個ﾓｰﾄﾞ
      ORB
      AND     M274  ; 締め部　位置決め 入り端
      AND     M17  ; 運転ﾓｰﾄﾞ切替
      AND     X0  ; 運転準備入り
      ANI     M287  ; 締め部　着座確認後退端
      OUT     M633  ; 締め部　着座確認 入り
3785  LD      M633  ; 締め部　着座確認 入り
      OUT     Y2EA  ; 締め部　着座確認 SOL
3787  LD      M421  ; 連続運転
      AND     T226  ; 締め部　ﾅｯﾄﾗﾝﾅｰ ﾊﾟﾚｯﾄ有り
      AND     L155  ; IAI締め部ﾜｰｸｾｯﾄ　完了
      ANI     M3000  ; 作業者ﾜｰｸ取出し
      ANI     L156  ; ﾅｯﾄﾗﾝﾅ　締め確認
      ANI     L1001  ; 締め動作無し　　記憶送り
      LD      M404  ; 各個実行
      AND     Y1187  ; 画面PBL締め部　ﾜｰｸ押え 押え
      ORB
      AND     M274  ; 締め部　位置決め 入り端
      LD      M640  ; 締め部　ﾜｰｸ押え 押え
      LD      M419  ; 初期SOL励磁
      AND     M276  ; 締め部　ﾜｰｸ押え 押え端
      ORB
      ANI     M641  ; 締め部　ﾜｰｸ押え 戻し
      ORB
      AND     M17  ; 運転ﾓｰﾄﾞ切替
      AND     X0  ; 運転準備入り
      OUT     M640  ; 締め部　ﾜｰｸ押え 押え
3806  LD      M421  ; 連続運転
      LD      L156  ; ﾅｯﾄﾗﾝﾅ　締め確認
      OR      M3000  ; 作業者ﾜｰｸ取出し
      ANB
      LD      M404  ; 各個実行
      AND     Y1186  ; 画面PBL締め部　ﾜｰｸ押え 戻し
      ORB
      OR      M300  ; 原点復帰PB
      LD      M641  ; 締め部　ﾜｰｸ押え 戻し
      LD      M419  ; 初期SOL励磁
      AND     M277  ; 締め部　ﾜｰｸ押え 戻し端
      ORB
      ANI     M640  ; 締め部　ﾜｰｸ押え 押え
      ORB
      AND     M17  ; 運転ﾓｰﾄﾞ切替
      AND     X0  ; 運転準備入り
      OUT     M641  ; 締め部　ﾜｰｸ押え 戻し
3823  LD      M640  ; 締め部　ﾜｰｸ押え 押え
      ANI     Y2F7  ; 締め部　ﾜｰｸ押え 戻し SOL
      OUT     Y2F6  ; 締め部　ﾜｰｸ押え 押えSOL
3826  LD      M641  ; 締め部　ﾜｰｸ押え 戻し
      ANI     Y2F6  ; 締め部　ﾜｰｸ押え 押えSOL
      OUT     Y2F7  ; 締め部　ﾜｰｸ押え 戻し SOL
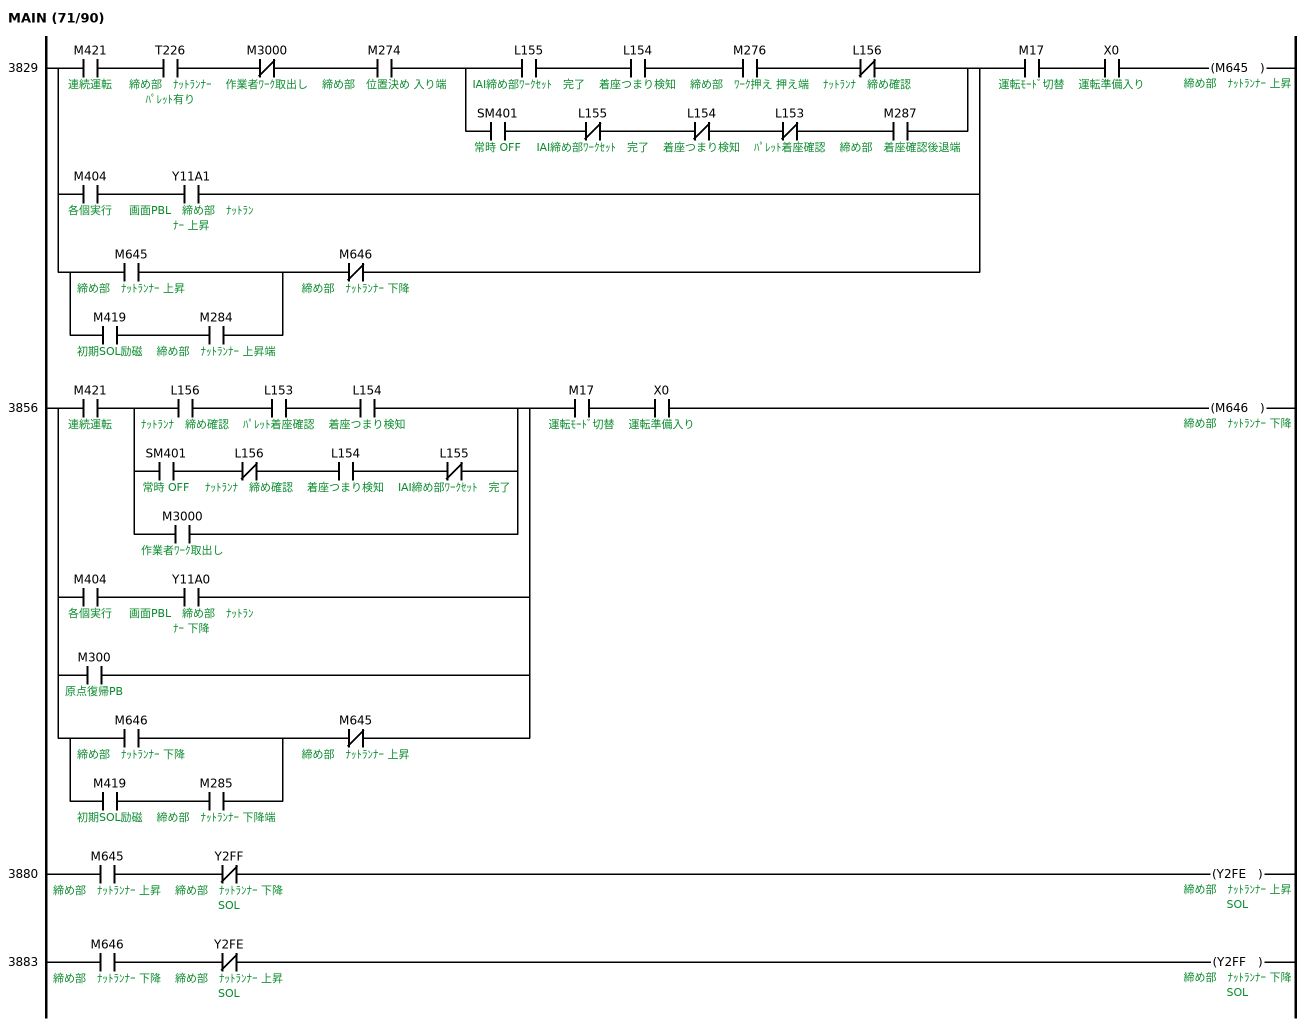
3829  LD      M421  ; 連続運転
      AND     T226  ; 締め部　ﾅｯﾄﾗﾝﾅｰ ﾊﾟﾚｯﾄ有り
      ANI     M3000  ; 作業者ﾜｰｸ取出し
      AND     M274  ; 締め部　位置決め 入り端
      LD      L155  ; IAI締め部ﾜｰｸｾｯﾄ　完了
      AND     L154  ; 着座つまり検知
      AND     M276  ; 締め部　ﾜｰｸ押え 押え端
      ANI     L156  ; ﾅｯﾄﾗﾝﾅ　締め確認
      LD      SM401  ; 常時 OFF
      ANI     L155  ; IAI締め部ﾜｰｸｾｯﾄ　完了
      ANI     L154  ; 着座つまり検知
      ANI     L153  ; ﾊﾟﾚｯﾄ着座確認
      AND     M287  ; 締め部　着座確認後退端
      ORB
      ANB
      LD      M404  ; 各個実行
      AND     Y11A1  ; 画面PBL　締め部　ﾅｯﾄﾗﾝﾅｰ 上昇
      ORB
      LD      M645  ; 締め部　ﾅｯﾄﾗﾝﾅｰ 上昇
      LD      M419  ; 初期SOL励磁
      AND     M284  ; 締め部　ﾅｯﾄﾗﾝﾅｰ 上昇端
      ORB
      ANI     M646  ; 締め部　ﾅｯﾄﾗﾝﾅｰ 下降
      ORB
      AND     M17  ; 運転ﾓｰﾄﾞ切替
      AND     X0  ; 運転準備入り
      OUT     M645  ; 締め部　ﾅｯﾄﾗﾝﾅｰ 上昇
3856  LD      M421  ; 連続運転
      LD      L156  ; ﾅｯﾄﾗﾝﾅ　締め確認
      AND     L153  ; ﾊﾟﾚｯﾄ着座確認
      AND     L154  ; 着座つまり検知
      LD      SM401  ; 常時 OFF
      ANI     L156  ; ﾅｯﾄﾗﾝﾅ　締め確認
      AND     L154  ; 着座つまり検知
      ANI     L155  ; IAI締め部ﾜｰｸｾｯﾄ　完了
      ORB
      OR      M3000  ; 作業者ﾜｰｸ取出し
      ANB
      LD      M404  ; 各個実行
      AND     Y11A0  ; 画面PBL　締め部　ﾅｯﾄﾗﾝﾅｰ 下降
      ORB
      OR      M300  ; 原点復帰PB
      LD      M646  ; 締め部　ﾅｯﾄﾗﾝﾅｰ 下降
      LD      M419  ; 初期SOL励磁
      AND     M285  ; 締め部　ﾅｯﾄﾗﾝﾅｰ 下降端
      ORB
      ANI     M645  ; 締め部　ﾅｯﾄﾗﾝﾅｰ 上昇
      ORB
      AND     M17  ; 運転ﾓｰﾄﾞ切替
      AND     X0  ; 運転準備入り
      OUT     M646  ; 締め部　ﾅｯﾄﾗﾝﾅｰ 下降
3880  LD      M645  ; 締め部　ﾅｯﾄﾗﾝﾅｰ 上昇
      ANI     Y2FF  ; 締め部　ﾅｯﾄﾗﾝﾅｰ 下降 SOL
      OUT     Y2FE  ; 締め部　ﾅｯﾄﾗﾝﾅｰ 上昇 SOL
3883  LD      M646  ; 締め部　ﾅｯﾄﾗﾝﾅｰ 下降
      ANI     Y2FE  ; 締め部　ﾅｯﾄﾗﾝﾅｰ 上昇 SOL
      OUT     Y2FF  ; 締め部　ﾅｯﾄﾗﾝﾅｰ 下降 SOL
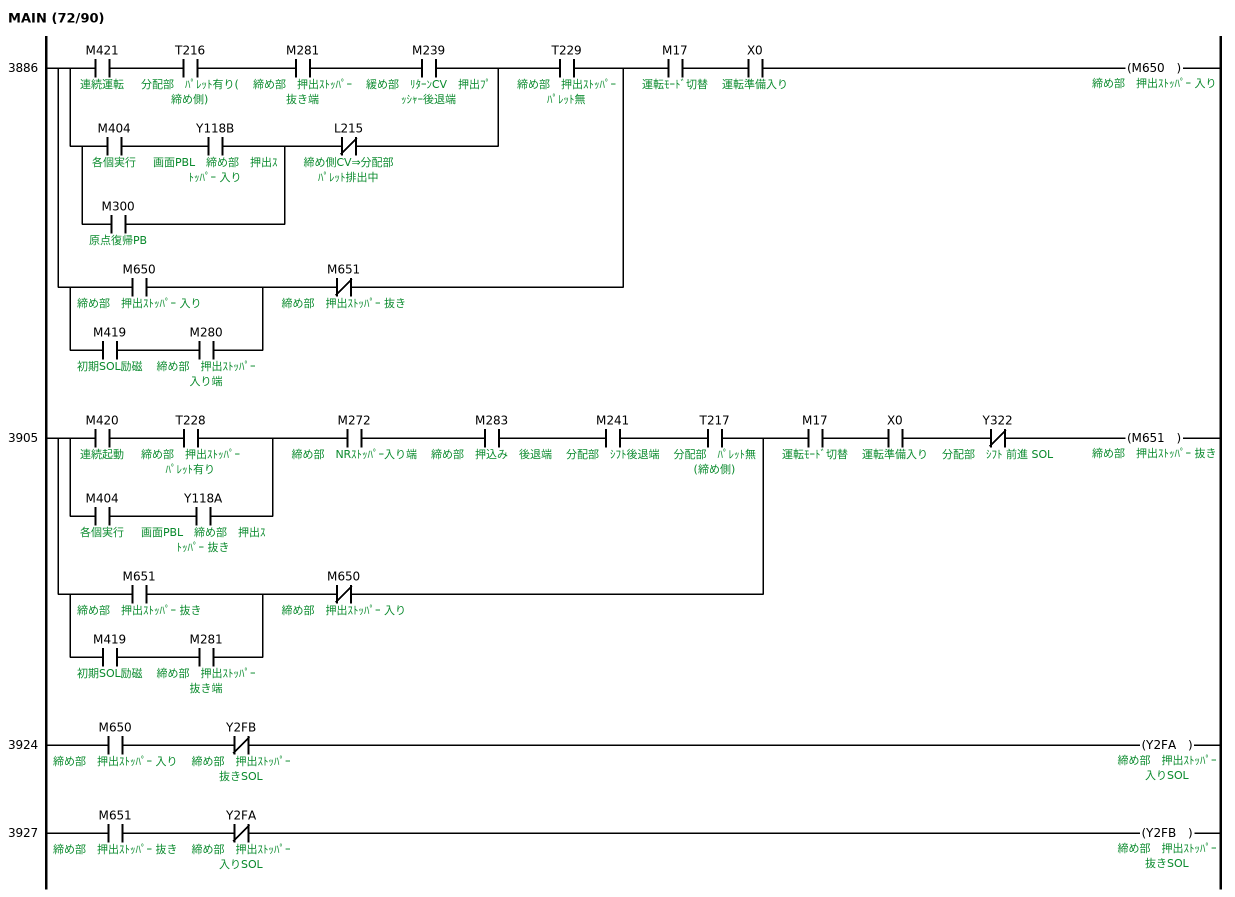
3886  LD      M421  ; 連続運転
      AND     T216  ; 分配部　ﾊﾟﾚｯﾄ有り(締め側)
      AND     M281  ; 締め部　押出ｽﾄｯﾊﾟｰ 抜き端
      AND     M239  ; 緩め部　ﾘﾀｰﾝCV　押出ﾌﾟｯｼｬｰ後退端
      LD      M404  ; 各個実行
      AND     Y118B  ; 画面PBL　締め部　押出ｽﾄｯﾊﾟｰ 入り
      OR      M300  ; 原点復帰PB
      ANI     L215  ; 締め側CV⇒分配部 ﾊﾟﾚｯﾄ排出中
      ORB
      AND     T229  ; 締め部　押出ｽﾄｯﾊﾟｰ ﾊﾟﾚｯﾄ無
      LD      M650  ; 締め部　押出ｽﾄｯﾊﾟｰ 入り
      LD      M419  ; 初期SOL励磁
      AND     M280  ; 締め部　押出ｽﾄｯﾊﾟｰ 入り端
      ORB
      ANI     M651  ; 締め部　押出ｽﾄｯﾊﾟｰ 抜き
      ORB
      AND     M17  ; 運転ﾓｰﾄﾞ切替
      AND     X0  ; 運転準備入り
      OUT     M650  ; 締め部　押出ｽﾄｯﾊﾟｰ 入り
3905  LD      M420  ; 連続起動
      AND     T228  ; 締め部　押出ｽﾄｯﾊﾟｰ ﾊﾟﾚｯﾄ有り
      LD      M404  ; 各個実行
      AND     Y118A  ; 画面PBL　締め部　押出ｽﾄｯﾊﾟｰ 抜き
      ORB
      AND     M272  ; 締め部　NRｽﾄｯﾊﾟｰ入り端
      AND     M283  ; 締め部　押込み　後退端
      AND     M241  ; 分配部　ｼﾌﾄ後退端
      AND     T217  ; 分配部　ﾊﾟﾚｯﾄ無 (締め側)
      LD      M651  ; 締め部　押出ｽﾄｯﾊﾟｰ 抜き
      LD      M419  ; 初期SOL励磁
      AND     M281  ; 締め部　押出ｽﾄｯﾊﾟｰ 抜き端
      ORB
      ANI     M650  ; 締め部　押出ｽﾄｯﾊﾟｰ 入り
      ORB
      AND     M17  ; 運転ﾓｰﾄﾞ切替
      AND     X0  ; 運転準備入り
      ANI     Y322  ; 分配部　ｼﾌﾄ 前進 SOL
      OUT     M651  ; 締め部　押出ｽﾄｯﾊﾟｰ 抜き
3924  LD      M650  ; 締め部　押出ｽﾄｯﾊﾟｰ 入り
      ANI     Y2FB  ; 締め部　押出ｽﾄｯﾊﾟｰ 抜きSOL
      OUT     Y2FA  ; 締め部　押出ｽﾄｯﾊﾟｰ 入りSOL
3927  LD      M651  ; 締め部　押出ｽﾄｯﾊﾟｰ 抜き
      ANI     Y2FA  ; 締め部　押出ｽﾄｯﾊﾟｰ 入りSOL
      OUT     Y2FB  ; 締め部　押出ｽﾄｯﾊﾟｰ 抜きSOL
